# B&R Automation Studio project NAELD004C00R10L518F00 (part 14)

#### Act_OptP0934RstMnl.st
```iecst
ACTION Act_OptP0934RstMnl:

	IF EDGEPOS((bManualMod = FALSE) OR (p_eAWOpenStatus = Error)) THEN

		eAWOpenAct	:= AWActIdle;

		bJogSlow				:= FALSE;
		bJogFast				:= FALSE;
		fbJogSlowToFastDlyTm.IN	:= FALSE;

		tyP0934AW.tyAW.tyBtnGo.bRtCompl					:= FALSE;
		tyP0934AW.tyAW.tyBtnGo.bValue					:= FALSE;
		tyP0934AW.tyAW.tyBtnGo.bRtLk					:= FALSE;
		tyP0934AW.tyAW.tyBtnGo.uiMaskRtStat.0			:= FALSE;

		tyP0934AW.tyMotionStd.tyBtnPwr.bRtCompl				:= FALSE;
		tyP0934AW.tyMotionStd.tyBtnStop.bRtCompl			:= FALSE;
		tyP0934AW.tyMotionStd.tyBtnOrigin.bRtCompl			:= FALSE;
		tyP0934AW.tyMotionStd.tyBtnRst.bRtCompl				:= FALSE;
		tyP0934AW.tyMotionStd.tyBtnMovAbs.bRtCompl			:= FALSE;
		tyP0934AW.tyMotionStd.tyBtnMovRel.bRtCompl			:= FALSE;
		tyP0934AW.tyMotionStd.tyBtnJogOpen.bRtCompl			:= FALSE;
		tyP0934AW.tyMotionStd.tyBtnJogClose.bRtCompl		:= FALSE;

		tyP0934AW.tyMotionStd.tyBtnPwr.bValue				:= FALSE;
		tyP0934AW.tyMotionStd.tyBtnStop.bValue				:= TRUE;
		tyP0934AW.tyMotionStd.tyBtnOrigin.bValue			:= FALSE;
		tyP0934AW.tyMotionStd.tyBtnRst.bValue				:= FALSE;
		tyP0934AW.tyMotionStd.tyBtnMovAbs.bValue			:= FALSE;
		tyP0934AW.tyMotionStd.tyBtnMovRel.bValue			:= FALSE;
		tyP0934AW.tyMotionStd.tyBtnJogOpen.bValue			:= FALSE;
		tyP0934AW.tyMotionStd.tyBtnJogClose.bValue			:= FALSE;

		tyP0934AW.tyMotionStd.tyBtnPwr.bRtLk				:= FALSE;
		tyP0934AW.tyMotionStd.tyBtnStop.bRtLk				:= TRUE;
		tyP0934AW.tyMotionStd.tyBtnOrigin.bRtLk				:= FALSE;
		tyP0934AW.tyMotionStd.tyBtnRst.bRtLk				:= FALSE;
		tyP0934AW.tyMotionStd.tyBtnMovAbs.bRtLk				:= FALSE;
		tyP0934AW.tyMotionStd.tyBtnMovRel.bRtLk				:= FALSE;
		tyP0934AW.tyMotionStd.tyBtnJogOpen.bRtLk			:= FALSE;
		tyP0934AW.tyMotionStd.tyBtnJogClose.bRtLk			:= FALSE;

		tyP0934AW.tyMotionStd.tyBtnPwr.uiMaskRtStat			:= TRUE;
		tyP0934AW.tyMotionStd.tyBtnOrigin.uiMaskRtStat		:= FALSE;
		tyP0934AW.tyMotionStd.tyBtnRst.uiMaskRtStat			:= TRUE;
		tyP0934AW.tyMotionStd.tyBtnMovAbs.uiMaskRtStat		:= FALSE;
		tyP0934AW.tyMotionStd.tyBtnMovRel.uiMaskRtStat		:= FALSE;
		tyP0934AW.tyMotionStd.tyBtnJogOpen.uiMaskRtStat		:= FALSE;
		tyP0934AW.tyMotionStd.tyBtnJogClose.uiMaskRtStat	:= FALSE;

	END_IF

	eInShutterAct	:= PneuActIdle;
	eOutShutterAct	:= PneuActIdle;

	tyP0934AW.tyInOutletShutterFB.tyBtnClose.bRtCompl	:= FALSE;
	tyP0934AW.tyInOutletShutterFB.tyBtnClose.bValue	:= FALSE;
	tyP0934AW.tyInOutletShutterFB.tyBtnOpen.bRtCompl	:= FALSE;
	tyP0934AW.tyInOutletShutterFB.tyBtnOpen.bValue	:= FALSE;

END_ACTION
```

#### Act_OptP0934UpdtDat.st
```iecst
ACTION Act_OptP0934UpdtDat:

	tyP0934AW.tyMotionStd.tyNumCurrPos.diValue			:= p_diAWOpenActualPos;
	tyP0934AW.tyMotionStd.tyNumErrCode.diValue			:= UDINT_TO_DINT(p_udiAWOpenAxisErrID);
	tyP0934AW.tyMotionStd.tyBitmapPwr.usiValueIdx		:= BOOL_TO_USINT(p_bAWOpenPwrOn);
	tyP0934AW.tyMotionStd.tyBitmapRst.usiValueIdx		:= BOOL_TO_USINT(NOT p_bAWOpenAxisErr);
	tyP0934AW.tyMotionStd.tyBitmapOrigin.usiValueIdx	:= BOOL_TO_USINT(p_bAWOpenIsHomed);
	tyP0934AW.tyMotionStd.tyBtnOpenLmtSen.bValue		:= p_bAWOpenOpenSen;
	tyP0934AW.tyMotionStd.tyBtnCloseLmtSen.bValue		:= p_bAWOpenCloseSen;

	//Machine Bitmap //0open ,1close
	IF p_bAWOpenIsHomed = TRUE THEN
		IF p_diAWOpenActualPos <= (p_tyNtParamCurr.tyProdRcpWidth.diMax / 2) THEN
			tyP0934AW.tyMotionStd.tyBitmapMc.uiValueIdx 	:= 0;
		ELSE
			tyP0934AW.tyMotionStd.tyBitmapMc.uiValueIdx 	:= 1;
		END_IF
	ELSE
		tyP0934AW.tyMotionStd.tyBitmapMc.uiValueIdx	:= 0;
	END_IF

	IF p_tyNtParamCurr.eProjMag = LDMagTriple AND p_tyNtParamCurr.bMagAutoVerifyPrep = FALSE AND p_tyNtParamCurr.bProjMotorizedPullerPrep = FALSE AND p_tyNtParamCurr.bProjTopToBtmDefault = TRUE THEN
		IF 	tyP0934AW.tyMotionStd.tyBitmapMc.uiValueIdx < 200 THEN
			tyP0934AW.tyMotionStd.tyBitmapMc.uiValueIdx	:= tyP0934AW.tyMotionStd.tyBitmapMc.uiValueIdx + 200;
		END_IF
	ELSIF p_tyNtParamCurr.eProjMag = LDMagTriple AND p_tyNtParamCurr.bMagAutoVerifyPrep = FALSE AND p_tyNtParamCurr.bProjMotorizedPullerPrep = FALSE AND p_tyNtParamCurr.bProjTopToBtmDefault = FALSE THEN
			IF 	tyP0934AW.tyMotionStd.tyBitmapMc.uiValueIdx < 200 THEN
				tyP0934AW.tyMotionStd.tyBitmapMc.uiValueIdx	:= tyP0934AW.tyMotionStd.tyBitmapMc.uiValueIdx + 426;
			END_IF

	ELSIF p_tyNtParamCurr.eProjMag = LDMagDual AND p_tyNtParamCurr.bMagAutoVerifyPrep = FALSE THEN
		IF 	tyP0934AW.tyMotionStd.tyBitmapMc.uiValueIdx < 100 THEN
			IF p_tyNtParamCurr.sJobNo = '2023-0258A01' THEN
				tyP0934AW.tyMotionStd.tyBitmapMc.uiValueIdx	:= tyP0934AW.tyMotionStd.tyBitmapMc.uiValueIdx + 450;
			ELSIF p_tyNtParamCurr.sJobNo = '2023-0276A01' THEN
				tyP0934AW.tyMotionStd.tyBitmapMc.uiValueIdx	:= tyP0934AW.tyMotionStd.tyBitmapMc.uiValueIdx + 480;
			ELSE
				tyP0934AW.tyMotionStd.tyBitmapMc.uiValueIdx	:= tyP0934AW.tyMotionStd.tyBitmapMc.uiValueIdx + 200;
			END_IF
		END_IF
	ELSIF  p_tyNtParamCurr.bMagAutoVerifyPrep = TRUE THEN
		IF 	tyP0934AW.tyMotionStd.tyBitmapMc.uiValueIdx < 200 THEN
			tyP0934AW.tyMotionStd.tyBitmapMc.uiValueIdx	:= tyP0934AW.tyMotionStd.tyBitmapMc.uiValueIdx + 426;
		END_IF

	ELSIF p_tyNtParamCurr.eProjMag = LDMagTriple AND p_tyNtParamCurr.bMagAutoVerifyPrep = FALSE AND p_tyNtParamCurr.bProjMotorizedPullerPrep = TRUE
		AND p_tyNtParamCurr.bProjPullerRotCylPrep = FALSE THEN //fix (siemens)
		IF 	tyP0934AW.tyMotionStd.tyBitmapMc.uiValueIdx < 340 THEN
			tyP0934AW.tyMotionStd.tyBitmapMc.uiValueIdx:= tyP0934AW.tyMotionStd.tyBitmapMc.uiValueIdx + 340;
		END_IF
	ELSIF  p_tyNtParamCurr.eProjMag = LDMagTriple AND p_tyNtParamCurr.bMagAutoVerifyPrep = FALSE AND p_tyNtParamCurr.bProjMotorizedPullerPrep = TRUE
		AND p_tyNtParamCurr.bProjCurtainSenPrep = FALSE THEN
		IF 	tyP0934AW.tyMotionStd.tyBitmapMc.uiValueIdx < 300 THEN
			tyP0934AW.tyMotionStd.tyBitmapMc.uiValueIdx:= tyP0934AW.tyMotionStd.tyBitmapMc.uiValueIdx + 300;
		END_IF
	ELSIF  p_tyNtParamCurr.eProjMag = LDMagTriple AND p_tyNtParamCurr.bMagAutoVerifyPrep = FALSE AND p_tyNtParamCurr.bProjMotorizedPullerPrep = TRUE
		AND p_tyNtParamCurr.bProjCurtainSenPrep = TRUE AND p_tyNtParamCurr.bProjTopToBtmDefault = TRUE THEN
		IF 	tyP0934AW.tyMotionStd.tyBitmapMc.uiValueIdx < 365 THEN
			tyP0934AW.tyMotionStd.tyBitmapMc.uiValueIdx:= tyP0934AW.tyMotionStd.tyBitmapMc.uiValueIdx + 365;
		END_IF
	ELSIF p_tyNtParamCurr.eProjMag = LDMagTriple AND p_tyNtParamCurr.bMagAutoVerifyPrep = FALSE AND p_tyNtParamCurr.bProjMotorizedPullerPrep = TRUE
		AND p_tyNtParamCurr.bProjCurtainSenPrep = TRUE AND p_tyNtParamCurr.bProjTopToBtmDefault = FALSE THEN
		IF  tyP0934AW.tyMotionStd.tyBitmapMc.uiValueIdx < 426 THEN
			tyP0934AW.tyMotionStd.tyBitmapMc.uiValueIdx	:= tyP0934AW.tyMotionStd.tyBitmapMc.uiValueIdx + 426;
		END_IF
	END_IF
END_ACTION
```

#### Act_EntP0935Disp.st
```iecst
ACTION Act_EntP0935Disp:

	//Access Address
	p_tyC0001MotionStd ACCESS ADR(tyP0935Lifter.tyMotionStd);

	p_tyC0002FullMask ACCESS ADR(tyP0935Lifter.tyFullMaskHide);

	p_tyC0004Navi ACCESS ADR(tyP0935Lifter.tyNaviBack);

	p_tyC0005Main ACCESS ADR(tyCommon.tyMain);

	p_tyC0007Notif ACCESS ADR(tyCommon.tyNotif);

	p_tyC0008MsgBox ACCESS ADR(tyP0935Lifter.tyMsgBoxHide);

	p_tyC0009Info ACCESS ADR(tyCommon.tyInfo);

	p_tyP0935Lifter ACCESS ADR(tyP0935Lifter.tyLifter);

	//Display
	tyP0935Lifter.tyMotionStd.tyBtnPwr.bValue	:= p_bLifterBtmPwrOn;

	IF p_tyNtParamCurr.bProjLifterMagPlatform = FALSE THEN
	//	tyP0935Lifter.tyLifter.tyNumNewSlt.diValueMax	:= p_tyMagRcpCurrRcp.diTtlSlt + 1;
		tyP0935Lifter.tyLifter.tyNumNewSlt.diValueMax	:= p_tyMagRcpCurrRcp.diTtlSlt;
		tyP0935Lifter.tyLifter.tyNumNewSlt.diValueMin	:= p_tyNtParamCurr.diProjMagMinSlt;
	ELSE
		tyP0935Lifter.tyLifter.tyNumNewSlt.diValueMax	:= p_tyMagRcpCurrRcp.diTtlSlt;
		tyP0935Lifter.tyLifter.tyNumNewSlt.diValueMin	:= p_tyNtParamCurr.diProjMagMinSlt;
	END_IF

END_ACTION
```

#### Act_OptP0935FBCtrl.st
```iecst
ACTION Act_OptP0935FBCtrl:

	fbJogSlowToFastDlyTm.PT	:= T#2s;
	fbJogSlowToFastDlyTm;
	fbLmtRstTm;

	//Lifter Safety Sensor Interruption
	IF EDGENEG(p_tyDI.bLifterSafetyLmtSW1 AND p_tyDI.bLifterSafetyLmtSW2 AND p_tyDI.bLifterTimingBeltSen) THEN
		tyP0935Lifter.tyMotionStd.tyBtnStop.bRtCompl	:= TRUE;
	END_IF

//	IF EDGEPOS((p_udiLifterBtmAxisErrID = 21570 OR p_udiLifterBtmAxisErrID = 21571)
	IF EDGEPOS((p_bLifterBtmFwdLmtSen OR p_bLifterBtmRevLmtSen OR p_udiLifterBtmAxisErrID = 21570 OR p_udiLifterBtmAxisErrID = 21571)
		AND tyP0935Lifter.tyMotionStd.tyBtnJogDown.bValue = FALSE
		AND tyP0935Lifter.tyMotionStd.tyBtnJogUp.bValue = FALSE)
	THEN
		fbLmtRstTm.IN				:= TRUE;
	END_IF

	IF fbLmtRstTm.Q = TRUE THEN
		tyP0935Lifter.tyMotionStd.tyBtnRst.bRtCompl		:= TRUE;
	END_IF

	IF (tyP0935Lifter.tyMotionStd.tyBtnJogUp.bValue = FALSE AND tyP0935Lifter.tyMotionStd.tyBtnJogDown.bValue = FALSE) AND (p_bLifterBtmJogging = TRUE) THEN
		bJogStopLifter	:= TRUE;
	END_IF

	IF tyP0935Lifter.tyMotionStd.tyBtnStop.bRtCompl = TRUE THEN
		eLifterBtmAct		:= LifterActStop;

		IF p_eLifterBtmStat = LifterActStop AND p_eLifterBtmStatus = Done THEN
			eLifterBtmAct	:= LifterActIdle;

			tyP0935Lifter.tyMotionStd.tyBtnStop.bRtCompl			:= FALSE;
			tyP0935Lifter.tyMotionStd.tyBtnJogDown.bRtCompl			:= FALSE;
			tyP0935Lifter.tyMotionStd.tyBtnJogUp.bRtCompl			:= FALSE;
			tyP0935Lifter.tyMotionStd.tyBtnOrigin.bRtCompl			:= FALSE;
			tyP0935Lifter.tyMotionStd.tyBtnMovAbs.bRtCompl			:= FALSE;
			tyP0935Lifter.tyMotionStd.tyBtnMovRel.bRtCompl			:= FALSE;
			tyP0935Lifter.tyLifter.tyBtnGo.bRtCompl					:= FALSE;
			tyP0935Lifter.tyLifter.tyBtnNxtSlt.bRtCompl				:= FALSE;
			tyP0935Lifter.tyLifter.tyBtnPrevSlt.bRtCompl			:= FALSE;
			tyP0935Lifter.tyLifter.tyBtnGoLaneA.bRtCompl			:= FALSE;
			tyP0935Lifter.tyLifter.tyBtnGoLaneB.bRtCompl			:= FALSE;

			tyP0935Lifter.tyMotionStd.tyBtnStop.bValue				:= TRUE;
			tyP0935Lifter.tyMotionStd.tyBtnJogDown.bValue			:= FALSE;
			tyP0935Lifter.tyMotionStd.tyBtnJogUp.bValue				:= FALSE;
			tyP0935Lifter.tyMotionStd.tyBtnOrigin.bValue			:= FALSE;
			tyP0935Lifter.tyMotionStd.tyBtnMovAbs.bValue			:= FALSE;
			tyP0935Lifter.tyMotionStd.tyBtnMovRel.bValue			:= FALSE;
			tyP0935Lifter.tyLifter.tyBtnGo.bValue					:= FALSE;
			tyP0935Lifter.tyLifter.tyBtnNxtSlt.bValue				:= FALSE;
			tyP0935Lifter.tyLifter.tyBtnPrevSlt.bValue				:= FALSE;
			tyP0935Lifter.tyLifter.tyBtnGoLaneA.bValue				:= FALSE;
			tyP0935Lifter.tyLifter.tyBtnGoLaneB.bValue				:= FALSE;

			tyP0935Lifter.tyMotionStd.tyBtnStop.bRtLk				:= TRUE;
			tyP0935Lifter.tyMotionStd.tyBtnJogDown.bRtLk			:= FALSE;
			tyP0935Lifter.tyMotionStd.tyBtnJogUp.bRtLk				:= FALSE;
			tyP0935Lifter.tyMotionStd.tyBtnOrigin.bRtLk				:= FALSE;
			tyP0935Lifter.tyMotionStd.tyBtnMovAbs.bRtLk				:= FALSE;
			tyP0935Lifter.tyMotionStd.tyBtnMovRel.bRtLk				:= FALSE;
			tyP0935Lifter.tyLifter.tyBtnGo.bRtLk					:= FALSE;
			tyP0935Lifter.tyLifter.tyBtnNxtSlt.bRtLk				:= FALSE;
			tyP0935Lifter.tyLifter.tyBtnPrevSlt.bRtLk				:= FALSE;
			tyP0935Lifter.tyLifter.tyBtnGoLaneA.bRtLk				:= FALSE;
			tyP0935Lifter.tyLifter.tyBtnGoLaneB.bRtLk				:= FALSE;
		END_IF

	ELSIF (tyP0935Lifter.tyMotionStd.tyBtnJogDown.bRtCompl = TRUE) OR (tyP0935Lifter.tyMotionStd.tyBtnJogUp.bRtCompl = TRUE) OR (bJogStopLifter = TRUE) THEN
		bJogSlow					:= FALSE;
		bJogFast					:= FALSE;
		fbJogSlowToFastDlyTm.IN		:= FALSE;

		eLifterBtmAct		:= LifterActJogStop;

		IF p_eLifterBtmStat = LifterActJogStop AND p_eLifterBtmStatus = Done THEN
			eLifterBtmAct		:= LifterActIdle;

			bJogStopLifter	:= FALSE;

			tyP0935Lifter.tyMotionStd.tyBtnStop.bRtCompl			:= FALSE;
			tyP0935Lifter.tyMotionStd.tyBtnJogDown.bRtCompl			:= FALSE;
			tyP0935Lifter.tyMotionStd.tyBtnJogUp.bRtCompl			:= FALSE;
			tyP0935Lifter.tyMotionStd.tyBtnOrigin.bRtCompl			:= FALSE;
			tyP0935Lifter.tyMotionStd.tyBtnMovAbs.bRtCompl			:= FALSE;
			tyP0935Lifter.tyMotionStd.tyBtnMovRel.bRtCompl			:= FALSE;
			tyP0935Lifter.tyLifter.tyBtnGo.bRtCompl					:= FALSE;
			tyP0935Lifter.tyLifter.tyBtnNxtSlt.bRtCompl				:= FALSE;
			tyP0935Lifter.tyLifter.tyBtnPrevSlt.bRtCompl			:= FALSE;
			tyP0935Lifter.tyLifter.tyBtnGoLaneA.bRtCompl 			:= FALSE;
			tyP0935Lifter.tyLifter.tyBtnGoLaneB.bRtCompl 			:= FALSE;

			tyP0935Lifter.tyMotionStd.tyBtnStop.bValue				:= TRUE;
			tyP0935Lifter.tyMotionStd.tyBtnJogDown.bValue			:= FALSE;
			tyP0935Lifter.tyMotionStd.tyBtnJogUp.bValue				:= FALSE;
			tyP0935Lifter.tyMotionStd.tyBtnOrigin.bValue			:= FALSE;
			tyP0935Lifter.tyMotionStd.tyBtnMovAbs.bValue			:= FALSE;
			tyP0935Lifter.tyMotionStd.tyBtnMovRel.bValue			:= FALSE;
			tyP0935Lifter.tyLifter.tyBtnGo.bValue					:= FALSE;
			tyP0935Lifter.tyLifter.tyBtnNxtSlt.bValue				:= FALSE;
			tyP0935Lifter.tyLifter.tyBtnPrevSlt.bValue				:= FALSE;
			tyP0935Lifter.tyLifter.tyBtnGoLaneA.bValue 				:= FALSE;
			tyP0935Lifter.tyLifter.tyBtnGoLaneB.bValue 				:= FALSE;

			tyP0935Lifter.tyMotionStd.tyBtnStop.bRtLk				:= TRUE;
			tyP0935Lifter.tyMotionStd.tyBtnJogDown.bRtLk			:= FALSE;
			tyP0935Lifter.tyMotionStd.tyBtnJogUp.bRtLk				:= FALSE;
			tyP0935Lifter.tyMotionStd.tyBtnOrigin.bRtLk				:= FALSE;
			tyP0935Lifter.tyMotionStd.tyBtnMovAbs.bRtLk				:= FALSE;
			tyP0935Lifter.tyMotionStd.tyBtnMovRel.bRtLk				:= FALSE;
			tyP0935Lifter.tyLifter.tyBtnGo.bRtLk					:= FALSE;
			tyP0935Lifter.tyLifter.tyBtnNxtSlt.bRtLk				:= FALSE;
			tyP0935Lifter.tyLifter.tyBtnPrevSlt.bRtLk				:= FALSE;
			tyP0935Lifter.tyLifter.tyBtnGoLaneA.bRtLk 				:= FALSE;
			tyP0935Lifter.tyLifter.tyBtnGoLaneB.bRtLk 				:= FALSE;

		END_IF

	ELSIF tyP0935Lifter.tyMotionStd.tyBtnPwr.bRtCompl = TRUE THEN
		tyP0935Lifter.tyMotionStd.tyBtnPwr.bRtLk					:= TRUE;

		IF tyP0935Lifter.tyMotionStd.tyBtnPwr.bValue = TRUE THEN
			eLifterBtmAct		:= LifterActPwrOn;

			IF p_eLifterBtmStat = LifterActPwrOn AND p_eLifterBtmStatus = Done THEN
				eLifterBtmAct	:= LifterActIdle;

				tyP0935Lifter.tyMotionStd.tyBtnPwr.bRtCompl		:= FALSE;
				tyP0935Lifter.tyMotionStd.tyBtnPwr.bRtLk		:= FALSE;
			END_IF
		ELSE
			eLifterBtmAct		:= LifterActPwrOff;

			IF p_eLifterBtmStat = LifterActPwrOff AND p_eLifterBtmStatus = Done THEN
				eLifterBtmAct	:= LifterActIdle;

				tyP0935Lifter.tyMotionStd.tyBtnPwr.bRtCompl		:= FALSE;
				tyP0935Lifter.tyMotionStd.tyBtnPwr.bRtLk		:= FALSE;
			END_IF
		END_IF

	ELSIF tyP0935Lifter.tyMotionStd.tyBtnOrigin.bRtCompl = TRUE THEN
		tyP0935Lifter.tyMotionStd.tyBtnOrigin.bValue				:= TRUE;
		tyP0935Lifter.tyMotionStd.tyBtnStop.bValue					:= FALSE;

		tyP0935Lifter.tyMotionStd.tyBtnOrigin.bRtLk					:= TRUE;
		tyP0935Lifter.tyMotionStd.tyBtnStop.bRtLk					:= FALSE;

		eLifterBtmAct		:= LifterActHoming;

		IF p_eLifterBtmStat = LifterActHoming AND p_eLifterBtmStatus = Done THEN
			eLifterBtmAct	:= LifterActIdle;

			tyP0935Lifter.tyMotionStd.tyBtnOrigin.bRtCompl		:= FALSE;
			tyP0935Lifter.tyMotionStd.tyBtnOrigin.bValue		:= FALSE;
			tyP0935Lifter.tyMotionStd.tyBtnStop.bValue			:= TRUE;

			tyP0935Lifter.tyMotionStd.tyBtnOrigin.bRtLk			:= FALSE;
			tyP0935Lifter.tyMotionStd.tyBtnStop.bRtLk			:= TRUE;

		END_IF

	ELSIF tyP0935Lifter.tyMotionStd.tyBtnRst.bRtCompl = TRUE THEN
		tyP0935Lifter.tyMotionStd.tyBtnRst.bValue				:= TRUE;
		tyP0935Lifter.tyMotionStd.tyBtnRst.bRtLk				:= TRUE;

		eLifterBtmAct		:= LifterActRstAxisErr;

		IF p_eLifterBtmStat = LifterActRstAxisErr AND p_eLifterBtmStatus = Done THEN
			eLifterBtmAct	:= LifterActIdle;

			tyP0935Lifter.tyMotionStd.tyBtnRst.bRtCompl			:= FALSE;
			tyP0935Lifter.tyMotionStd.tyBtnRst.bValue			:= FALSE;
			tyP0935Lifter.tyMotionStd.tyBtnRst.bRtLk			:= FALSE;

			fbLmtRstTm.IN			:= FALSE;
		END_IF

	ELSIF tyP0935Lifter.tyLifter.tyBtnGo.bRtCompl = TRUE THEN
		tyP0935Lifter.tyLifter.tyBtnGo.bValue				:= TRUE;
		tyP0935Lifter.tyMotionStd.tyBtnStop.bValue			:= FALSE;

		tyP0935Lifter.tyLifter.tyBtnGo.bRtLk				:= TRUE;
		tyP0935Lifter.tyMotionStd.tyBtnStop.bRtLk			:= FALSE;

		(*diMnlLifterMag1GoSlt	:= tyP0935Lifter.tyLifter.tyNumNewSlt.diValue;*)
		diMnlLifterNomSpd		:= tyP0935Lifter.tyMotionStd.tyNumNomSpd.diValue;

		CASE tyP0935Lifter.tyLifter.tyNumMagPos.diValue OF
			1:
				eLifterBtmAct	:= LifterActGoASltPos;
				diMnlLifterMag1GoSlt	:= tyP0935Lifter.tyLifter.tyNumNewSlt.diValue;

			2:
				eLifterBtmAct	:= LifterActGoBSltPos;
				diMnlLifterMag2GoSlt	:= tyP0935Lifter.tyLifter.tyNumNewSlt.diValue;

			3:
				eLifterBtmAct	:= LifterActGoCSltPos;
				diMnlLifterMag3GoSlt	:= tyP0935Lifter.tyLifter.tyNumNewSlt.diValue;

			4:
				eLifterBtmAct	:= LifterActGoDSltPos;
				diMnlLifterMag3GoSlt	:= tyP0935Lifter.tyLifter.tyNumNewSlt.diValue;
		END_CASE

		IF (p_eLifterBtmStat = LifterActGoASltPos
			OR p_eLifterBtmStat = LifterActGoBSltPos
			OR p_eLifterBtmStat = LifterActGoCSltPos
			OR p_eLifterBtmStat = LifterActGoDSltPos)
			AND p_eLifterBtmStatus = Done THEN
			eLifterBtmAct	:= LifterActIdle;

			tyP0935Lifter.tyLifter.tyBtnGo.bRtCompl				:= FALSE;
			tyP0935Lifter.tyLifter.tyBtnGo.bValue				:= FALSE;
			tyP0935Lifter.tyMotionStd.tyBtnStop.bValue			:= TRUE;

			tyP0935Lifter.tyLifter.tyBtnGo.bRtLk				:= FALSE;
			tyP0935Lifter.tyMotionStd.tyBtnStop.bRtLk			:= TRUE;
		END_IF

	ELSIF tyP0935Lifter.tyLifter.tyBtnNxtSlt.bRtCompl = TRUE THEN
		tyP0935Lifter.tyLifter.tyBtnNxtSlt.bValue				:= TRUE;
		tyP0935Lifter.tyMotionStd.tyBtnStop.bValue				:= FALSE;

		tyP0935Lifter.tyLifter.tyBtnNxtSlt.bRtLk				:= TRUE;
		tyP0935Lifter.tyMotionStd.tyBtnStop.bRtLk				:= FALSE;

		(*diMnlLifterMag1GoSlt	:= tyP0935Lifter.tyLifter.tyNumNewSlt.diValue;*)
		diMnlLifterNomSpd		:= tyP0935Lifter.tyMotionStd.tyNumNomSpd.diValue;

		CASE tyP0935Lifter.tyLifter.tyNumMagPos.diValue OF
			1:
				eLifterBtmAct	:= LifterActGoNxtASltPos;
				diMnlLifterMag1GoSlt	:= tyP0935Lifter.tyLifter.tyNumNewSlt.diValue;
			2:
				eLifterBtmAct	:= LifterActGoNxtBSltPos;
				diMnlLifterMag2GoSlt	:= tyP0935Lifter.tyLifter.tyNumNewSlt.diValue;
			3:
				eLifterBtmAct	:= LifterActGoNxtCSltPos;
				diMnlLifterMag3GoSlt	:= tyP0935Lifter.tyLifter.tyNumNewSlt.diValue;
			4:
				eLifterBtmAct	:= LifterActGoNxtDSltPos;
				diMnlLifterMag4GoSlt	:= tyP0935Lifter.tyLifter.tyNumNewSlt.diValue;

		END_CASE

		IF (p_eLifterBtmStat = LifterActGoNxtASltPos
			OR p_eLifterBtmStat = LifterActGoNxtBSltPos
			OR p_eLifterBtmStat = LifterActGoNxtCSltPos
			OR p_eLifterBtmStat = LifterActGoNxtDSltPos)
			AND p_eLifterBtmStatus = Done THEN
			eLifterBtmAct	:= LifterActIdle;

			tyP0935Lifter.tyLifter.tyBtnNxtSlt.bRtCompl				:= FALSE;
			tyP0935Lifter.tyLifter.tyBtnNxtSlt.bValue				:= FALSE;
			tyP0935Lifter.tyMotionStd.tyBtnStop.bValue				:= TRUE;

			tyP0935Lifter.tyLifter.tyBtnNxtSlt.bRtLk				:= FALSE;
			tyP0935Lifter.tyMotionStd.tyBtnStop.bRtLk				:= TRUE;
		END_IF

	ELSIF tyP0935Lifter.tyLifter.tyBtnPrevSlt.bRtCompl = TRUE THEN
		tyP0935Lifter.tyLifter.tyBtnPrevSlt.bValue				:= TRUE;
		tyP0935Lifter.tyMotionStd.tyBtnStop.bValue				:= FALSE;

		tyP0935Lifter.tyLifter.tyBtnPrevSlt.bRtLk				:= TRUE;
		tyP0935Lifter.tyMotionStd.tyBtnStop.bRtLk				:= FALSE;

		//diMnlLifterMag1GoSlt	:= tyP0935Lifter.tyLifter.tyNumNewSlt.diValue;
		diMnlLifterNomSpd		:= tyP0935Lifter.tyMotionStd.tyNumNomSpd.diValue;

		CASE tyP0935Lifter.tyLifter.tyNumMagPos.diValue OF

			1:
				eLifterBtmAct	:= LifterActGoPrevASltPos;
				diMnlLifterMag1GoSlt	:= tyP0935Lifter.tyLifter.tyNumNewSlt.diValue;

			2:
				eLifterBtmAct	:= LifterActGoPrevBSltPos;
				diMnlLifterMag2GoSlt	:= tyP0935Lifter.tyLifter.tyNumNewSlt.diValue;

			3:
				eLifterBtmAct	:= LifterActGoPrevCSltPos;
				diMnlLifterMag3GoSlt	:= tyP0935Lifter.tyLifter.tyNumNewSlt.diValue;

			4:
				eLifterBtmAct	:= LifterActGoPrevDSltPos;
				diMnlLifterMag4GoSlt	:= tyP0935Lifter.tyLifter.tyNumNewSlt.diValue;

		END_CASE

		IF (p_eLifterBtmStat = LifterActGoPrevASltPos
			OR p_eLifterBtmStat = LifterActGoPrevBSltPos
			OR p_eLifterBtmStat = LifterActGoPrevCSltPos
			OR p_eLifterBtmStat = LifterActGoPrevDSltPos)
			AND p_eLifterBtmStatus = Done THEN
			eLifterBtmAct	:= LifterActIdle;

			tyP0935Lifter.tyLifter.tyBtnPrevSlt.bRtCompl				:= FALSE;
			tyP0935Lifter.tyLifter.tyBtnPrevSlt.bValue					:= FALSE;
			tyP0935Lifter.tyMotionStd.tyBtnStop.bValue					:= TRUE;

			tyP0935Lifter.tyLifter.tyBtnPrevSlt.bRtLk					:= FALSE;
			tyP0935Lifter.tyMotionStd.tyBtnStop.bRtLk					:= TRUE;
		END_IF

	ELSIF tyP0935Lifter.tyLifter.tyBtnGoLaneA.bRtCompl = TRUE THEN
		tyP0935Lifter.tyLifter.tyBtnGoLaneA.bValue	:= TRUE;
		tyP0935Lifter.tyMotionStd.tyBtnStop.bValue	:= FALSE;

		tyP0935Lifter.tyLifter.tyBtnGoLaneA.bRtLk	:= TRUE;
		tyP0935Lifter.tyMotionStd.tyBtnStop.bRtLk	:= FALSE;

		diMnlLifterNomSpd	:= tyP0935Lifter.tyMotionStd.tyNumNomSpd.diValue;

		eLifterBtmAct	:= LifterActGoAPos;

		IF p_eLifterBtmStat = LifterActGoAPos AND p_eLifterBtmStatus = Done THEN
			eLifterBtmAct	:= LifterActIdle;

			tyP0935Lifter.tyLifter.tyBtnGoLaneA.bRtCompl	:= FALSE;

			tyP0935Lifter.tyLifter.tyBtnGoLaneA.bValue	:= FALSE;
			tyP0935Lifter.tyMotionStd.tyBtnStop.bValue	:= TRUE;

			tyP0935Lifter.tyLifter.tyBtnGoLaneA.bRtLk	:= FALSE;
			tyP0935Lifter.tyMotionStd.tyBtnStop.bRtLk	:= TRUE;
		END_IF

	ELSIF tyP0935Lifter.tyLifter.tyBtnGoLaneB.bRtCompl = TRUE THEN
		tyP0935Lifter.tyLifter.tyBtnGoLaneB.bValue	:= TRUE;
		tyP0935Lifter.tyMotionStd.tyBtnStop.bValue	:= FALSE;

		tyP0935Lifter.tyLifter.tyBtnGoLaneB.bRtLk	:= TRUE;
		tyP0935Lifter.tyMotionStd.tyBtnStop.bRtLk	:= FALSE;

		diMnlLifterNomSpd	:= tyP0935Lifter.tyMotionStd.tyNumNomSpd.diValue;

		eLifterBtmAct	:= LifterActGoBPos;

		IF p_eLifterBtmStat = LifterActGoBPos AND p_eLifterBtmStatus = Done THEN
			eLifterBtmAct	:= LifterActIdle;

			tyP0935Lifter.tyLifter.tyBtnGoLaneB.bRtCompl	:= FALSE;

			tyP0935Lifter.tyLifter.tyBtnGoLaneB.bValue	:= FALSE;
			tyP0935Lifter.tyMotionStd.tyBtnStop.bValue	:= TRUE;

			tyP0935Lifter.tyLifter.tyBtnGoLaneB.bRtLk	:= FALSE;
			tyP0935Lifter.tyMotionStd.tyBtnStop.bRtLk	:= TRUE;
		END_IF

	ELSIF tyP0935Lifter.tyMotionStd.tyBtnMovAbs.bRtCompl = TRUE THEN

		tyP0935Lifter.tyMotionStd.tyBtnMovAbs.bValue				:= TRUE;
		tyP0935Lifter.tyMotionStd.tyBtnStop.bValue					:= FALSE;

		tyP0935Lifter.tyMotionStd.tyBtnMovAbs.bRtLk					:= TRUE;
		tyP0935Lifter.tyMotionStd.tyBtnStop.bRtLk					:= FALSE;

		diMnlLifterTargetPos	:= tyP0935Lifter.tyMotionStd.tyNumTargetPos.diValue;
		diMnlLifterNomSpd		:= tyP0935Lifter.tyMotionStd.tyNumNomSpd.diValue;

		eLifterBtmAct			:= LifterActMovAbs;

		IF p_eLifterBtmStat = LifterActMovAbs AND p_eLifterBtmStatus = Done THEN
			eLifterBtmAct	:= LifterActIdle;

			tyP0935Lifter.tyMotionStd.tyBtnMovAbs.bRtCompl		:= FALSE;
			tyP0935Lifter.tyMotionStd.tyBtnMovAbs.bValue		:= FALSE;
			tyP0935Lifter.tyMotionStd.tyBtnStop.bValue			:= TRUE;

			tyP0935Lifter.tyMotionStd.tyBtnMovAbs.bRtLk			:= FALSE;
			tyP0935Lifter.tyMotionStd.tyBtnStop.bRtLk			:= TRUE;
		END_IF

	ELSIF tyP0935Lifter.tyMotionStd.tyBtnMovRel.bRtCompl = TRUE THEN
		tyP0935Lifter.tyMotionStd.tyBtnMovRel.bValue			:= TRUE;
		tyP0935Lifter.tyMotionStd.tyBtnStop.bValue				:= FALSE;

		tyP0935Lifter.tyMotionStd.tyBtnMovRel.bRtLk				:= TRUE;
		tyP0935Lifter.tyMotionStd.tyBtnStop.bRtLk				:= FALSE;

		diMnlLifterStepSize		:= tyP0935Lifter.tyMotionStd.tyNumStepSize.diValue;
		diMnlLifterNomSpd		:= tyP0935Lifter.tyMotionStd.tyNumNomSpd.diValue;

		eLifterBtmAct		:= LifterActMovRel;

		IF p_eLifterBtmStat = LifterActMovRel AND p_eLifterBtmStatus = Done THEN
			eLifterBtmAct	:= LifterActIdle;

			tyP0935Lifter.tyMotionStd.tyBtnMovRel.bRtCompl		:= FALSE;
			tyP0935Lifter.tyMotionStd.tyBtnMovRel.bValue		:= FALSE;
			tyP0935Lifter.tyMotionStd.tyBtnStop.bValue			:= TRUE;

			tyP0935Lifter.tyMotionStd.tyBtnMovRel.bRtLk			:= FALSE;
			tyP0935Lifter.tyMotionStd.tyBtnStop.bRtLk			:= TRUE;

		END_IF

	ELSIF (tyP0935Lifter.tyMotionStd.tyBtnJogDown.bValue = TRUE) AND (fbJogSlowToFastDlyTm.Q = FALSE) AND (bJogSlow = FALSE) THEN
		tyP0935Lifter.tyMotionStd.tyBtnStop.bValue				:= FALSE;
		tyP0935Lifter.tyMotionStd.tyBtnStop.bRtLk				:= FALSE;

		fbJogSlowToFastDlyTm.IN		:= TRUE;

		diMnlLifterJogSpd	:= tyP0935Lifter.tyMotionStd.tyNumSlwSpd.diValue;

		eLifterBtmAct		:= LifterActJogDown;

		IF p_eLifterBtmStat = LifterActJogDown AND p_eLifterBtmStatus = Done THEN

			eLifterBtmAct	:= LifterActIdle;
			bJogSlow				:= TRUE;

		ELSIF p_eLifterBtmStatus = Error THEN

			fbJogSlowToFastDlyTm.IN	:= FALSE;
			bJogSlow				:= TRUE;

		END_IF

	ELSIF (tyP0935Lifter.tyMotionStd.tyBtnJogDown.bValue = TRUE) AND (fbJogSlowToFastDlyTm.Q = TRUE) AND (bJogFast = FALSE) THEN
		tyP0935Lifter.tyMotionStd.tyBtnStop.bValue					:= FALSE;
		tyP0935Lifter.tyMotionStd.tyBtnStop.bRtLk					:= FALSE;

		fbJogSlowToFastDlyTm.IN		:= TRUE;

		diMnlLifterJogSpd	:= tyP0935Lifter.tyMotionStd.tyNumNomSpd.diValue;

		eLifterBtmAct		:= LifterActJogDown;

		IF p_eLifterBtmStat = LifterActJogDown AND p_eLifterBtmStatus = Done THEN
			eLifterBtmAct	:= LifterActIdle;
			bJogFast				:= TRUE;
		ELSIF p_eLifterBtmStatus = Error THEN
			fbJogSlowToFastDlyTm.IN	:= FALSE;
			bJogFast				:= TRUE;
		END_IF

	ELSIF (tyP0935Lifter.tyMotionStd.tyBtnJogUp.bValue = TRUE) AND (fbJogSlowToFastDlyTm.Q = FALSE) AND (bJogSlow = FALSE) THEN
		tyP0935Lifter.tyMotionStd.tyBtnStop.bValue				:= FALSE;
		tyP0935Lifter.tyMotionStd.tyBtnStop.bRtLk				:= FALSE;

		fbJogSlowToFastDlyTm.IN		:= TRUE;

		diMnlLifterJogSpd	:= tyP0935Lifter.tyMotionStd.tyNumSlwSpd.diValue;

		eLifterBtmAct		:= LifterActJogUp;

		IF p_eLifterBtmStat = LifterActJogUp AND p_eLifterBtmStatus = Done THEN
			eLifterBtmAct	:= LifterActIdle;
			bJogSlow				:= TRUE;

		ELSIF p_eLifterBtmStatus = Error THEN
			fbJogSlowToFastDlyTm.IN	:= FALSE;
			bJogSlow				:= TRUE;
		END_IF

	ELSIF (tyP0935Lifter.tyMotionStd.tyBtnJogUp.bValue = TRUE) AND (fbJogSlowToFastDlyTm.Q = TRUE) AND (bJogFast = FALSE) THEN

		tyP0935Lifter.tyMotionStd.tyBtnStop.bValue				:= FALSE;
		tyP0935Lifter.tyMotionStd.tyBtnStop.bRtLk				:= FALSE;

		fbJogSlowToFastDlyTm.IN		:= TRUE;

		diMnlLifterJogSpd	:= tyP0935Lifter.tyMotionStd.tyNumNomSpd.diValue;

		eLifterBtmAct		:= LifterActJogUp;

		IF p_eLifterBtmStat = LifterActJogUp AND p_eLifterBtmStatus = Done THEN
			eLifterBtmAct	:= LifterActIdle;
			bJogFast	:= TRUE;

		ELSIF p_eLifterBtmStatus = Error THEN
			fbJogSlowToFastDlyTm.IN	:= FALSE;
			bJogFast				:= TRUE;
		END_IF
	END_IF

	//Shutter Control
	IF tyP0935Lifter.tyInOutletShutterFB.tyBtnOpen.bRtCompl = TRUE THEN
		tyP0935Lifter.tyInOutletShutterFB.tyBtnOpen.bRtCompl	:= FALSE;

		tyP0935Lifter.tyInOutletShutterFB.tyBtnOpen.bValue	:= TRUE;
		tyP0935Lifter.tyInOutletShutterFB.tyBtnClose.bValue	:= FALSE;

	ELSIF tyP0935Lifter.tyInOutletShutterFB.tyBtnClose.bRtCompl = TRUE THEN
		tyP0935Lifter.tyInOutletShutterFB.tyBtnClose.bRtCompl	:= FALSE;

		tyP0935Lifter.tyInOutletShutterFB.tyBtnClose.bValue	:= TRUE;
		tyP0935Lifter.tyInOutletShutterFB.tyBtnOpen.bValue	:= FALSE;
	END_IF

	IF tyP0935Lifter.tyInOutletShutterFB.tyBtnOpen.bValue = TRUE THEN
		eInShutterAct	:= PneuActRet;
		eOutShutterAct	:= PneuActRet;

		IF (p_eInShutterStat = PneuActRet AND p_eInShutterStatus = Done)
			AND (p_eOutShutterStat = PneuActRet AND p_eOutShutterStatus = Done)
			THEN
			eInShutterAct	:= PneuActIdle;
			eOutShutterAct	:= PneuActIdle;
			tyP0935Lifter.tyInOutletShutterFB.tyBtnOpen.bValue	:= FALSE;
		ELSIF p_eInShutterStatus = Error OR p_eOutShutterStatus = Error THEN
			tyP0935Lifter.tyInOutletShutterFB.tyBtnOpen.bValue	:= FALSE;
		END_IF

	ELSIF tyP0935Lifter.tyInOutletShutterFB.tyBtnClose.bValue = TRUE THEN
		eInShutterAct	:= PneuActExt;
		eOutShutterAct	:= PneuActExt;
		IF (p_eInShutterStat = PneuActExt AND p_eInShutterStatus = Done)
			AND (p_eOutShutterStat = PneuActExt AND p_eOutShutterStatus = Done)
			THEN
			eInShutterAct	:= PneuActIdle;
			eOutShutterAct	:= PneuActIdle;
			tyP0935Lifter.tyInOutletShutterFB.tyBtnClose.bValue := FALSE;
		ELSIF p_eInShutterStatus = Error OR p_eOutShutterStatus = Error THEN
			tyP0935Lifter.tyInOutletShutterFB.tyBtnClose.bValue := FALSE;
		END_IF
	END_IF

END_ACTION
```

#### Act_OptP0935FullMask.st
```iecst
ACTION Act_OptP0935FullMask:

	IF eCurrPage = UIP0935Lifter THEN

		IF p_tyDI.bEStopSig = FALSE THEN
			p_tyC0002FullMask ACCESS ADR(tyP0935Lifter.tyFullMaskEStop);

		ELSIF p_tyDI.bCoverSWSig = FALSE THEN
			p_tyC0002FullMask ACCESS ADR(tyP0935Lifter.tyFullMaskCWSig);

		ELSIF p_tyDI.bSafetyRlySig = FALSE THEN
			p_tyC0002FullMask ACCESS ADR(tyP0935Lifter.tyFullMaskSafetyRly);

		ELSIF p_tyDI.bPullerRetRS = FALSE THEN
			p_tyC0002FullMask ACCESS ADR(tyP0935Lifter.tyFullMaskPullInterrupt);

		ELSIF p_tyNtParamCurr.bProjInletShutPrep AND (p_tyDI.bInShutterCloseRS = FALSE
			OR (p_tyDI.bInShutterCloseRS2 = FALSE AND p_tyNtParamCurr.tyDISettings.diInShutterCloseRS2 > 0)
			OR (p_tyDI.bInShutterCloseRS3 = FALSE AND p_tyNtParamCurr.tyDISettings.diInShutterCloseRS3 > 0)) THEN
			IF p_tyNtParamCurr.bProjCurtainSenPrep THEN
				IF p_tyDI.bInShutterCloseRS = FALSE OR p_tyDI.bInShutterCloseRS2 = FALSE OR p_tyDI.bInShutterCloseRS3 = FALSE THEN
					p_tyC0002FullMask ACCESS ADR(tyP0935Lifter.tyFullMaskInShutOpnInterrupt);
				END_IF
			ELSE
				IF p_tyDI.bInShutterCloseRS = FALSE THEN
					p_tyC0002FullMask ACCESS ADR(tyP0935Lifter.tyFullMaskInShutOpnInterrupt);
				END_IF
			END_IF

	//	ELSIF p_tyNtParamCurr.bProjOutletShutPrep AND p_tyDI.bOutShutterCloseRS = FALSE AND p_McParamOutShutterDis = FALSE THEN
		ELSIF p_tyNtParamCurr.bProjOutletShutPrep AND p_tyDI.bOutShutterCloseRS = FALSE THEN
			p_tyC0002FullMask ACCESS ADR(tyP0935Lifter.tyFullMaskOutShutOpnInterrupt);

		ELSIF p_tyDI.bConvLftSen THEN
			p_tyC0002FullMask ACCESS ADR(tyP0935Lifter.tyFullMaskLftSenInterrupt);

		ELSIF p_tyDI.bConvRgtSen THEN
			p_tyC0002FullMask ACCESS ADR(tyP0935Lifter.tyFullMaskRgtSenInterrupt);

		ELSIF p_tyDI.bLifterSafetyLmtSW1 = FALSE OR p_tyDI.bLifterSafetyLmtSW2 = FALSE THEN
			p_tyC0002FullMask ACCESS ADR(tyP0935Lifter.tyFullMaskSafetyLmtSW);

		ELSIF p_tyDI.bLifterTimingBeltSen = FALSE THEN
			p_tyC0002FullMask ACCESS ADR(tyP0935Lifter.tyFullMaskTimingBelt);

		ELSE
			p_tyC0002FullMask ACCESS ADR(tyP0935Lifter.tyFullMaskHide);

		END_IF

	END_IF

END_ACTION
```

#### Act_OptP0935Keypad.st
```iecst
ACTION Act_OptP0935Keypad:

	IF fUIOutRtStatTPIsOpen(ADR(tyP0935Lifter.tyMotionStd.tyNumTargetPos.uiRtStat)) = TRUE THEN
		tyProperty.tyKeypad.tyStringTitle.sKeypadTitle	:= tyP0935Lifter.tyMotionStd.tyNumTargetPos.sKeypadTitle;

	ELSIF fUIOutRtStatTPIsOpen(ADR(tyP0935Lifter.tyMotionStd.tyNumStepSize.uiRtStat)) = TRUE THEN
		tyProperty.tyKeypad.tyStringTitle.sKeypadTitle	:= tyP0935Lifter.tyMotionStd.tyNumStepSize.sKeypadTitle;

	ELSIF fUIOutRtStatTPIsOpen(ADR(tyP0935Lifter.tyMotionStd.tyNumNomSpd.uiRtStat)) = TRUE THEN
		tyProperty.tyKeypad.tyStringTitle.sKeypadTitle	:= tyP0935Lifter.tyMotionStd.tyNumNomSpd.sKeypadTitle;

	ELSIF fUIOutRtStatTPIsOpen(ADR(tyP0935Lifter.tyMotionStd.tyNumSlwSpd.uiRtStat)) = TRUE THEN
		tyProperty.tyKeypad.tyStringTitle.sKeypadTitle	:= tyP0935Lifter.tyMotionStd.tyNumSlwSpd.sKeypadTitle;

	ELSIF fUIOutRtStatTPIsOpen(ADR(tyP0935Lifter.tyLifter.tyNumNewSlt.uiRtStat)) = TRUE THEN
		tyProperty.tyKeypad.tyStringTitle.sKeypadTitle	:= tyP0935Lifter.tyLifter.tyNumNewSlt.sKeypadTitle;

	ELSIF fUIOutRtStatTPIsOpen(ADR(tyP0935Lifter.tyLifter.tyNumMagPos.uiRtStat)) = TRUE THEN
		tyProperty.tyKeypad.tyStringTitle.sKeypadTitle	:= tyP0935Lifter.tyLifter.tyNumMagPos.sKeypadTitle;

	END_IF

END_ACTION
```

#### Act_OptP0935Mask.st
```iecst
ACTION Act_OptP0935Mask:

	// Interlock Power
	IF p_bLifterBtmAxisErr = TRUE AND p_bLifterBtmPwrOn = FALSE THEN
		fUIInRtStatOff(ADR(tyP0935Lifter.tyMotionStd.tyBtnPwr.uiMaskRtStat));
		tyP0935Lifter.tyMotionStd.tyBtnPwr.bValue		:= FALSE;
	ELSE
		fUIInRtStatHide(ADR(tyP0935Lifter.tyMotionStd.tyBtnPwr.uiMaskRtStat));
	END_IF

	// Interlock Others Move
	IF p_bLifterBtmAxisErr = TRUE OR p_bLifterBtmPwrOn = FALSE THEN
		fUIInRtStatOff(ADR(tyP0935Lifter.tyMotionStd.tyBtnOrigin.uiMaskRtStat));
		fUIInRtStatOff(ADR(tyP0935Lifter.tyMotionStd.tyBtnMovRel.uiMaskRtStat));
		fUIInRtStatOff(ADR(tyP0935Lifter.tyMotionStd.tyBtnJogUp.uiMaskRtStat));
		fUIInRtStatOff(ADR(tyP0935Lifter.tyMotionStd.tyBtnJogDown.uiMaskRtStat));
	ELSE
		fUIInRtStatHide(ADR(tyP0935Lifter.tyMotionStd.tyBtnOrigin.uiMaskRtStat));
		fUIInRtStatHide(ADR(tyP0935Lifter.tyMotionStd.tyBtnMovRel.uiMaskRtStat));
		fUIInRtStatHide(ADR(tyP0935Lifter.tyMotionStd.tyBtnJogUp.uiMaskRtStat));
		fUIInRtStatHide(ADR(tyP0935Lifter.tyMotionStd.tyBtnJogDown.uiMaskRtStat));
	END_IF

	// Interlock Move Absolute
	IF p_bLifterBtmAxisErr = TRUE OR p_bLifterBtmPwrOn = FALSE OR p_bLifterBtmIsHomed = FALSE THEN

		fUIInRtStatOff(ADR(tyP0935Lifter.tyMotionStd.tyBtnMovAbs.uiMaskRtStat));

		fUIInRtStatOff(ADR(tyP0935Lifter.tyLifter.tyBtnGo.uiMaskRtStat));
		fUIInRtStatOff(ADR(tyP0935Lifter.tyLifter.tyBtnNxtSlt.uiMaskRtStat));
		fUIInRtStatOff(ADR(tyP0935Lifter.tyLifter.tyBtnPrevSlt.uiMaskRtStat));
		fUIInRtStatOff(ADR(tyP0935Lifter.tyLifter.tyBtnGoLaneA.uiMaskRtStat));
		fUIInRtStatOff(ADR(tyP0935Lifter.tyLifter.tyBtnGoLaneB.uiMaskRtStat));

	ELSE
		fUIInRtStatHide(ADR(tyP0935Lifter.tyMotionStd.tyBtnMovAbs.uiMaskRtStat));

		fUIInRtStatHide(ADR(tyP0935Lifter.tyLifter.tyBtnGo.uiMaskRtStat));
		fUIInRtStatHide(ADR(tyP0935Lifter.tyLifter.tyBtnNxtSlt.uiMaskRtStat));
		fUIInRtStatHide(ADR(tyP0935Lifter.tyLifter.tyBtnPrevSlt.uiMaskRtStat));
		fUIInRtStatHide(ADR(tyP0935Lifter.tyLifter.tyBtnGoLaneA.uiMaskRtStat));
		fUIInRtStatHide(ADR(tyP0935Lifter.tyLifter.tyBtnGoLaneB.uiMaskRtStat));

	END_IF

	//Interlock Limit Sensor
	IF tyP0935Lifter.tyMotionStd.tyBtnDownLmtSen.bValue = TRUE THEN
		fUIInRtStatOff(ADR(tyP0935Lifter.tyMotionStd.tyBtnJogDown.uiMaskRtStat));
	END_IF

	IF tyP0935Lifter.tyMotionStd.tyBtnUpLmtSen.bValue = TRUE THEN
		fUIInRtStatOff(ADR(tyP0935Lifter.tyMotionStd.tyBtnJogUp.uiMaskRtStat));
	END_IF

	// Interlock When Moving
	IF tyP0935Lifter.tyMotionStd.tyBtnOrigin.bRtCompl = TRUE THEN

		fUIInRtStatOff(ADR(tyP0935Lifter.tyMotionStd.tyBtnMovAbs.uiMaskRtStat));
		fUIInRtStatOff(ADR(tyP0935Lifter.tyMotionStd.tyBtnMovRel.uiMaskRtStat));
		fUIInRtStatOff(ADR(tyP0935Lifter.tyMotionStd.tyBtnJogUp.uiMaskRtStat));
		fUIInRtStatOff(ADR(tyP0935Lifter.tyMotionStd.tyBtnJogDown.uiMaskRtStat));

		fUIInRtStatOff(ADR(tyP0935Lifter.tyLifter.tyBtnGo.uiMaskRtStat));
		fUIInRtStatOff(ADR(tyP0935Lifter.tyLifter.tyBtnPrevSlt.uiMaskRtStat));
		fUIInRtStatOff(ADR(tyP0935Lifter.tyLifter.tyBtnNxtSlt.uiMaskRtStat));
		fUIInRtStatOff(ADR(tyP0935Lifter.tyLifter.tyBtnGoLaneA.uiMaskRtStat));
		fUIInRtStatOff(ADR(tyP0935Lifter.tyLifter.tyBtnGoLaneB.uiMaskRtStat));

	ELSIF tyP0935Lifter.tyMotionStd.tyBtnMovAbs.bRtCompl = TRUE THEN

		fUIInRtStatOff(ADR(tyP0935Lifter.tyMotionStd.tyBtnOrigin.uiMaskRtStat));
		fUIInRtStatOff(ADR(tyP0935Lifter.tyMotionStd.tyBtnMovRel.uiMaskRtStat));
		fUIInRtStatOff(ADR(tyP0935Lifter.tyMotionStd.tyBtnJogUp.uiMaskRtStat));
		fUIInRtStatOff(ADR(tyP0935Lifter.tyMotionStd.tyBtnJogDown.uiMaskRtStat));

		fUIInRtStatOff(ADR(tyP0935Lifter.tyLifter.tyBtnGo.uiMaskRtStat));
		fUIInRtStatOff(ADR(tyP0935Lifter.tyLifter.tyBtnPrevSlt.uiMaskRtStat));
		fUIInRtStatOff(ADR(tyP0935Lifter.tyLifter.tyBtnNxtSlt.uiMaskRtStat));
		fUIInRtStatOff(ADR(tyP0935Lifter.tyLifter.tyBtnGoLaneA.uiMaskRtStat));
		fUIInRtStatOff(ADR(tyP0935Lifter.tyLifter.tyBtnGoLaneB.uiMaskRtStat));

	ELSIF tyP0935Lifter.tyMotionStd.tyBtnMovRel.bRtCompl = TRUE THEN

		fUIInRtStatOff(ADR(tyP0935Lifter.tyMotionStd.tyBtnOrigin.uiMaskRtStat));
		fUIInRtStatOff(ADR(tyP0935Lifter.tyMotionStd.tyBtnMovAbs.uiMaskRtStat));
		fUIInRtStatOff(ADR(tyP0935Lifter.tyMotionStd.tyBtnJogUp.uiMaskRtStat));
		fUIInRtStatOff(ADR(tyP0935Lifter.tyMotionStd.tyBtnJogDown.uiMaskRtStat));

		fUIInRtStatOff(ADR(tyP0935Lifter.tyLifter.tyBtnGo.uiMaskRtStat));
		fUIInRtStatOff(ADR(tyP0935Lifter.tyLifter.tyBtnNxtSlt.uiMaskRtStat));
		fUIInRtStatOff(ADR(tyP0935Lifter.tyLifter.tyBtnPrevSlt.uiMaskRtStat));
		fUIInRtStatOff(ADR(tyP0935Lifter.tyLifter.tyBtnGoLaneA.uiMaskRtStat));
		fUIInRtStatOff(ADR(tyP0935Lifter.tyLifter.tyBtnGoLaneB.uiMaskRtStat));

	ELSIF tyP0935Lifter.tyMotionStd.tyBtnJogDown.bRtCompl = TRUE OR tyP0935Lifter.tyMotionStd.tyBtnJogDown.bValue = TRUE THEN
		fUIInRtStatOff(ADR(tyP0935Lifter.tyMotionStd.tyBtnOrigin.uiMaskRtStat));
		fUIInRtStatOff(ADR(tyP0935Lifter.tyMotionStd.tyBtnMovAbs.uiMaskRtStat));
		fUIInRtStatOff(ADR(tyP0935Lifter.tyMotionStd.tyBtnMovRel.uiMaskRtStat));
		fUIInRtStatOff(ADR(tyP0935Lifter.tyMotionStd.tyBtnJogUp.uiMaskRtStat));

		fUIInRtStatOff(ADR(tyP0935Lifter.tyLifter.tyBtnGo.uiMaskRtStat));
		fUIInRtStatOff(ADR(tyP0935Lifter.tyLifter.tyBtnNxtSlt.uiMaskRtStat));
		fUIInRtStatOff(ADR(tyP0935Lifter.tyLifter.tyBtnPrevSlt.uiMaskRtStat));
		fUIInRtStatOff(ADR(tyP0935Lifter.tyLifter.tyBtnGoLaneA.uiMaskRtStat));
		fUIInRtStatOff(ADR(tyP0935Lifter.tyLifter.tyBtnGoLaneB.uiMaskRtStat));

	ELSIF tyP0935Lifter.tyMotionStd.tyBtnJogUp.bRtCompl = TRUE OR tyP0935Lifter.tyMotionStd.tyBtnJogUp.bValue = TRUE THEN
		fUIInRtStatOff(ADR(tyP0935Lifter.tyMotionStd.tyBtnOrigin.uiMaskRtStat));
		fUIInRtStatOff(ADR(tyP0935Lifter.tyMotionStd.tyBtnMovAbs.uiMaskRtStat));
		fUIInRtStatOff(ADR(tyP0935Lifter.tyMotionStd.tyBtnMovRel.uiMaskRtStat));
		fUIInRtStatOff(ADR(tyP0935Lifter.tyMotionStd.tyBtnJogDown.uiMaskRtStat));

		fUIInRtStatOff(ADR(tyP0935Lifter.tyLifter.tyBtnGo.uiMaskRtStat));
		fUIInRtStatOff(ADR(tyP0935Lifter.tyLifter.tyBtnNxtSlt.uiMaskRtStat));
		fUIInRtStatOff(ADR(tyP0935Lifter.tyLifter.tyBtnPrevSlt.uiMaskRtStat));
		fUIInRtStatOff(ADR(tyP0935Lifter.tyLifter.tyBtnGoLaneA.uiMaskRtStat));
		fUIInRtStatOff(ADR(tyP0935Lifter.tyLifter.tyBtnGoLaneB.uiMaskRtStat));

	ELSIF tyP0935Lifter.tyLifter.tyBtnGo.bRtCompl = TRUE THEN
		fUIInRtStatOff(ADR(tyP0935Lifter.tyMotionStd.tyBtnOrigin.uiMaskRtStat));
		fUIInRtStatOff(ADR(tyP0935Lifter.tyMotionStd.tyBtnMovAbs.uiMaskRtStat));
		fUIInRtStatOff(ADR(tyP0935Lifter.tyMotionStd.tyBtnMovRel.uiMaskRtStat));
		fUIInRtStatOff(ADR(tyP0935Lifter.tyMotionStd.tyBtnJogUp.uiMaskRtStat));
		fUIInRtStatOff(ADR(tyP0935Lifter.tyMotionStd.tyBtnJogDown.uiMaskRtStat));

		fUIInRtStatOff(ADR(tyP0935Lifter.tyLifter.tyBtnNxtSlt.uiMaskRtStat));
		fUIInRtStatOff(ADR(tyP0935Lifter.tyLifter.tyBtnPrevSlt.uiMaskRtStat));
		fUIInRtStatOff(ADR(tyP0935Lifter.tyLifter.tyBtnGoLaneA.uiMaskRtStat));
		fUIInRtStatOff(ADR(tyP0935Lifter.tyLifter.tyBtnGoLaneB.uiMaskRtStat));

	ELSIF tyP0935Lifter.tyLifter.tyBtnNxtSlt.bRtCompl = TRUE THEN
		fUIInRtStatOff(ADR(tyP0935Lifter.tyMotionStd.tyBtnOrigin.uiMaskRtStat));
		fUIInRtStatOff(ADR(tyP0935Lifter.tyMotionStd.tyBtnMovAbs.uiMaskRtStat));
		fUIInRtStatOff(ADR(tyP0935Lifter.tyMotionStd.tyBtnMovRel.uiMaskRtStat));
		fUIInRtStatOff(ADR(tyP0935Lifter.tyMotionStd.tyBtnJogUp.uiMaskRtStat));
		fUIInRtStatOff(ADR(tyP0935Lifter.tyMotionStd.tyBtnJogDown.uiMaskRtStat));

		fUIInRtStatOff(ADR(tyP0935Lifter.tyLifter.tyBtnGo.uiMaskRtStat));
		fUIInRtStatOff(ADR(tyP0935Lifter.tyLifter.tyBtnPrevSlt.uiMaskRtStat));
		fUIInRtStatOff(ADR(tyP0935Lifter.tyLifter.tyBtnGoLaneA.uiMaskRtStat));
		fUIInRtStatOff(ADR(tyP0935Lifter.tyLifter.tyBtnGoLaneB.uiMaskRtStat));

	ELSIF tyP0935Lifter.tyLifter.tyBtnPrevSlt.bRtCompl = TRUE THEN
		fUIInRtStatOff(ADR(tyP0935Lifter.tyMotionStd.tyBtnOrigin.uiMaskRtStat));
		fUIInRtStatOff(ADR(tyP0935Lifter.tyMotionStd.tyBtnMovAbs.uiMaskRtStat));
		fUIInRtStatOff(ADR(tyP0935Lifter.tyMotionStd.tyBtnMovRel.uiMaskRtStat));
		fUIInRtStatOff(ADR(tyP0935Lifter.tyMotionStd.tyBtnJogUp.uiMaskRtStat));
		fUIInRtStatOff(ADR(tyP0935Lifter.tyMotionStd.tyBtnJogDown.uiMaskRtStat));

		fUIInRtStatOff(ADR(tyP0935Lifter.tyLifter.tyBtnGo.uiMaskRtStat));
		fUIInRtStatOff(ADR(tyP0935Lifter.tyLifter.tyBtnNxtSlt.uiMaskRtStat));
		fUIInRtStatOff(ADR(tyP0935Lifter.tyLifter.tyBtnGoLaneA.uiMaskRtStat));
		fUIInRtStatOff(ADR(tyP0935Lifter.tyLifter.tyBtnGoLaneB.uiMaskRtStat));

	ELSIF tyP0935Lifter.tyLifter.tyBtnGoLaneA.bRtCompl = TRUE THEN
		fUIInRtStatOff(ADR(tyP0935Lifter.tyMotionStd.tyBtnOrigin.uiMaskRtStat));
		fUIInRtStatOff(ADR(tyP0935Lifter.tyMotionStd.tyBtnMovAbs.uiMaskRtStat));
		fUIInRtStatOff(ADR(tyP0935Lifter.tyMotionStd.tyBtnMovRel.uiMaskRtStat));
		fUIInRtStatOff(ADR(tyP0935Lifter.tyMotionStd.tyBtnJogUp.uiMaskRtStat));
		fUIInRtStatOff(ADR(tyP0935Lifter.tyMotionStd.tyBtnJogDown.uiMaskRtStat));

		fUIInRtStatOff(ADR(tyP0935Lifter.tyLifter.tyBtnGo.uiMaskRtStat));
		fUIInRtStatOff(ADR(tyP0935Lifter.tyLifter.tyBtnNxtSlt.uiMaskRtStat));
		fUIInRtStatOff(ADR(tyP0935Lifter.tyLifter.tyBtnPrevSlt.uiMaskRtStat));
		fUIInRtStatOff(ADR(tyP0935Lifter.tyLifter.tyBtnGoLaneB.uiMaskRtStat));

	ELSIF tyP0935Lifter.tyLifter.tyBtnGoLaneB.bRtCompl = TRUE THEN
		fUIInRtStatOff(ADR(tyP0935Lifter.tyMotionStd.tyBtnOrigin.uiMaskRtStat));
		fUIInRtStatOff(ADR(tyP0935Lifter.tyMotionStd.tyBtnMovAbs.uiMaskRtStat));
		fUIInRtStatOff(ADR(tyP0935Lifter.tyMotionStd.tyBtnMovRel.uiMaskRtStat));
		fUIInRtStatOff(ADR(tyP0935Lifter.tyMotionStd.tyBtnJogUp.uiMaskRtStat));
		fUIInRtStatOff(ADR(tyP0935Lifter.tyMotionStd.tyBtnJogDown.uiMaskRtStat));

		fUIInRtStatOff(ADR(tyP0935Lifter.tyLifter.tyBtnGo.uiMaskRtStat));
		fUIInRtStatOff(ADR(tyP0935Lifter.tyLifter.tyBtnNxtSlt.uiMaskRtStat));
		fUIInRtStatOff(ADR(tyP0935Lifter.tyLifter.tyBtnPrevSlt.uiMaskRtStat));
		fUIInRtStatOff(ADR(tyP0935Lifter.tyLifter.tyBtnGoLaneA.uiMaskRtStat));

	END_IF

	//Axis Error
	IF tyP0935Lifter.tyMotionStd.tyBtnPwr.bRtCompl = TRUE THEN
		fUIInRtStatOff(ADR(tyP0935Lifter.tyMotionStd.tyBtnRst.uiMaskRtStat));
	ELSE
		fUIInRtStatHide(ADR(tyP0935Lifter.tyMotionStd.tyBtnRst.uiMaskRtStat));
	END_IF

	//Next Slot
	IF p_diLifterBtmCurrSltA >= p_tyProdRcpCurrRcp0.diMaxSltValue THEN
		fUIInRtStatOff(ADR(tyP0935Lifter.tyLifter.tyBtnNxtSlt.uiMaskRtStat));
	END_IF

	//Previous Slot
	IF p_diLifterBtmCurrSltA <= p_tyProdRcpCurrRcp0.diMinSltValue THEN
		fUIInRtStatOff(ADR(tyP0935Lifter.tyLifter.tyBtnPrevSlt.uiMaskRtStat));
	END_IF

END_ACTION
```

#### Act_OptP0935RstMnl.st
```iecst
ACTION Act_OptP0935RstMnl:

	IF EDGEPOS((bManualMod = FALSE) OR (p_eLifterBtmStatus = Error)) THEN

		eLifterBtmAct	:= LifterActIdle;

		bJogSlow				:= FALSE;
		bJogFast				:= FALSE;
		fbJogSlowToFastDlyTm.IN	:= FALSE;

		tyP0935Lifter.tyLifter.tyBtnGo.bRtCompl					:= FALSE;
		tyP0935Lifter.tyLifter.tyBtnNxtSlt.bRtCompl				:= FALSE;
		tyP0935Lifter.tyLifter.tyBtnPrevSlt.bRtCompl			:= FALSE;
		tyP0935Lifter.tyLifter.tyBtnGoLaneA.bRtCompl			:= FALSE;
		tyP0935Lifter.tyLifter.tyBtnGoLaneB.bRtCompl			:= FALSE;

		tyP0935Lifter.tyLifter.tyBtnGo.bValue					:= FALSE;
		tyP0935Lifter.tyLifter.tyBtnNxtSlt.bValue				:= FALSE;
		tyP0935Lifter.tyLifter.tyBtnPrevSlt.bValue				:= FALSE;
		tyP0935Lifter.tyLifter.tyBtnGoLaneA.bValue				:= FALSE;
		tyP0935Lifter.tyLifter.tyBtnGoLaneB.bValue				:= FALSE;

		tyP0935Lifter.tyLifter.tyBtnGo.bRtLk					:= FALSE;
		tyP0935Lifter.tyLifter.tyBtnNxtSlt.bRtLk				:= FALSE;
		tyP0935Lifter.tyLifter.tyBtnPrevSlt.bRtLk				:= FALSE;
		tyP0935Lifter.tyLifter.tyBtnGoLaneA.bRtLk				:= FALSE;
		tyP0935Lifter.tyLifter.tyBtnGoLaneB.bRtLk				:= FALSE;

		tyP0935Lifter.tyLifter.tyBtnGo.uiMaskRtStat.0			:= FALSE;
		tyP0935Lifter.tyLifter.tyBtnNxtSlt.uiMaskRtStat.0		:= FALSE;
		tyP0935Lifter.tyLifter.tyBtnPrevSlt.uiMaskRtStat.0		:= FALSE;
		tyP0935Lifter.tyLifter.tyBtnGoLaneA.uiMaskRtStat.0		:= FALSE;
		tyP0935Lifter.tyLifter.tyBtnGoLaneB.uiMaskRtStat.0		:= FALSE;

		tyP0935Lifter.tyMotionStd.tyBtnPwr.bRtCompl				:= FALSE;
		tyP0935Lifter.tyMotionStd.tyBtnStop.bRtCompl			:= FALSE;
		tyP0935Lifter.tyMotionStd.tyBtnOrigin.bRtCompl			:= FALSE;
		tyP0935Lifter.tyMotionStd.tyBtnRst.bRtCompl				:= FALSE;
		tyP0935Lifter.tyMotionStd.tyBtnMovAbs.bRtCompl			:= FALSE;
		tyP0935Lifter.tyMotionStd.tyBtnMovRel.bRtCompl			:= FALSE;
		tyP0935Lifter.tyMotionStd.tyBtnJogUp.bRtCompl			:= FALSE;
		tyP0935Lifter.tyMotionStd.tyBtnJogDown.bRtCompl			:= FALSE;

		tyP0935Lifter.tyMotionStd.tyBtnPwr.bValue				:= FALSE;
		tyP0935Lifter.tyMotionStd.tyBtnStop.bValue				:= TRUE;
		tyP0935Lifter.tyMotionStd.tyBtnOrigin.bValue			:= FALSE;
		tyP0935Lifter.tyMotionStd.tyBtnRst.bValue				:= FALSE;
		tyP0935Lifter.tyMotionStd.tyBtnMovAbs.bValue			:= FALSE;
		tyP0935Lifter.tyMotionStd.tyBtnMovRel.bValue			:= FALSE;
		tyP0935Lifter.tyMotionStd.tyBtnJogUp.bValue				:= FALSE;
		tyP0935Lifter.tyMotionStd.tyBtnJogDown.bValue			:= FALSE;

		tyP0935Lifter.tyMotionStd.tyBtnPwr.bRtLk				:= FALSE;
		tyP0935Lifter.tyMotionStd.tyBtnStop.bRtLk				:= TRUE;
		tyP0935Lifter.tyMotionStd.tyBtnOrigin.bRtLk				:= FALSE;
		tyP0935Lifter.tyMotionStd.tyBtnRst.bRtLk				:= FALSE;
		tyP0935Lifter.tyMotionStd.tyBtnMovAbs.bRtLk				:= FALSE;
		tyP0935Lifter.tyMotionStd.tyBtnMovRel.bRtLk				:= FALSE;
		tyP0935Lifter.tyMotionStd.tyBtnJogUp.bRtLk				:= FALSE;
		tyP0935Lifter.tyMotionStd.tyBtnJogDown.bRtLk			:= FALSE;

		tyP0935Lifter.tyMotionStd.tyBtnPwr.uiMaskRtStat			:= TRUE;
		tyP0935Lifter.tyMotionStd.tyBtnOrigin.uiMaskRtStat		:= FALSE;
		tyP0935Lifter.tyMotionStd.tyBtnRst.uiMaskRtStat			:= TRUE;
		tyP0935Lifter.tyMotionStd.tyBtnMovAbs.uiMaskRtStat		:= FALSE;
		tyP0935Lifter.tyMotionStd.tyBtnMovRel.uiMaskRtStat		:= FALSE;
		tyP0935Lifter.tyMotionStd.tyBtnJogUp.uiMaskRtStat		:= FALSE;
		tyP0935Lifter.tyMotionStd.tyBtnJogDown.uiMaskRtStat		:= FALSE;

	END_IF

	eInShutterAct	:= PneuActIdle;
	eOutShutterAct	:= PneuActIdle;

	tyP0935Lifter.tyInOutletShutterFB.tyBtnClose.bRtCompl	:= FALSE;
	tyP0935Lifter.tyInOutletShutterFB.tyBtnClose.bValue	:= FALSE;
	tyP0935Lifter.tyInOutletShutterFB.tyBtnOpen.bRtCompl	:= FALSE;
	tyP0935Lifter.tyInOutletShutterFB.tyBtnOpen.bValue	:= FALSE;

END_ACTION
```

#### Act_OptP0935UpdtDat.st
```iecst
ACTION Act_OptP0935UpdtDat:

	tyP0935Lifter.tyMotionStd.tyNumCurrPos.diValue			:= p_diLifterBtmActualPos;
	tyP0935Lifter.tyMotionStd.tyNumErrCode.diValue			:= UDINT_TO_DINT(p_udiLifterBtmAxisErrID);
	tyP0935Lifter.tyMotionStd.tyBitmapPwr.usiValueIdx		:= BOOL_TO_USINT(p_bLifterBtmPwrOn);
	tyP0935Lifter.tyMotionStd.tyBitmapRst.usiValueIdx		:= BOOL_TO_USINT(NOT p_bLifterBtmAxisErr);
	tyP0935Lifter.tyMotionStd.tyBitmapOrigin.usiValueIdx	:= BOOL_TO_USINT(p_bLifterBtmIsHomed);
	tyP0935Lifter.tyMotionStd.tyBtnUpLmtSen.bValue			:= p_bLifterBtmUpSen;
	tyP0935Lifter.tyMotionStd.tyBtnDownLmtSen.bValue		:= p_bLifterBtmDownSen;

	//Machine Bitmap //default:2dn 3mid 4top
	IF  (p_tyNtParamCurr.eProjMag = LDMagDual)
		OR (p_tyNtParamCurr.eProjMag = LDMagTriple AND p_tyNtParamCurr.bMagAutoVerifyPrep = FALSE)
		THEN
			IF p_bLifterBtmIsHomed = TRUE THEN

					IF p_diLifterBtmActualPos <= (p_tyNtParamCurr.tyUILifterTargetPos.diMax / 3) THEN
						tyP0935Lifter.tyMotionStd.tyBitmapMc.uiValueIdx 	:= 2;
					ELSIF p_diLifterBtmActualPos <= (p_tyNtParamCurr.tyUILifterTargetPos.diMax / 3 * 2) THEN
						tyP0935Lifter.tyMotionStd.tyBitmapMc.uiValueIdx 	:= 3;
					ELSE
						tyP0935Lifter.tyMotionStd.tyBitmapMc.uiValueIdx 	:= 4;
					END_IF

			ELSE
				tyP0935Lifter.tyMotionStd.tyBitmapMc.uiValueIdx	:= 2;
			END_IF

	ELSIF p_tyNtParamCurr.eProjMag = LDMagTriple AND p_tyNtParamCurr.bMagAutoVerifyPrep = TRUE
		THEN
			IF p_bLifterBtmIsHomed = TRUE THEN

				IF p_diLifterBtmActualPos <= (p_tyNtParamCurr.tyUILifterTargetPos.diMax / 3) THEN
					tyP0935Lifter.tyMotionStd.tyBitmapMc.uiValueIdx 	:= 23;
				ELSIF p_diLifterBtmActualPos <= (p_tyNtParamCurr.tyUILifterTargetPos.diMax / 3 * 2) THEN
					tyP0935Lifter.tyMotionStd.tyBitmapMc.uiValueIdx 	:= 24;
				ELSE
					tyP0935Lifter.tyMotionStd.tyBitmapMc.uiValueIdx 	:= 25;
				END_IF

			ELSE
				tyP0935Lifter.tyMotionStd.tyBitmapMc.uiValueIdx	:= 23;
		END_IF
	ELSIF p_tyNtParamCurr.eProjMag = LDMagQuadruple AND p_tyNtParamCurr.bMagAutoVerifyPrep = TRUE
		THEN
		IF p_bLifterBtmIsHomed = TRUE THEN

			IF p_diLifterBtmActualPos <= (p_tyNtParamCurr.tyUILifterTargetPos.diMax / 3) THEN
				tyP0935Lifter.tyMotionStd.tyBitmapMc.uiValueIdx 	:= 27;
			ELSIF p_diLifterBtmActualPos <= (p_tyNtParamCurr.tyUILifterTargetPos.diMax / 3 * 2) THEN
				tyP0935Lifter.tyMotionStd.tyBitmapMc.uiValueIdx 	:= 28;
			ELSE
				tyP0935Lifter.tyMotionStd.tyBitmapMc.uiValueIdx 	:= 29;
			END_IF

		ELSE
			tyP0935Lifter.tyMotionStd.tyBitmapMc.uiValueIdx	:= 27;
		END_IF
	END_IF

	IF p_tyNtParamCurr.eProjMag = LDMagTriple AND p_tyNtParamCurr.bProjLifterMagPlatform THEN
		IF 	tyP0935Lifter.tyMotionStd.tyBitmapMc.uiValueIdx < 400 THEN
			tyP0935Lifter.tyMotionStd.tyBitmapMc.uiValueIdx	:= tyP0935Lifter.tyMotionStd.tyBitmapMc.uiValueIdx + 400;
		END_IF

	ELSIF p_tyNtParamCurr.eProjMag = LDMagTriple AND p_tyNtParamCurr.bMagAutoVerifyPrep = FALSE AND p_tyNtParamCurr.bProjMotorizedPullerPrep = FALSE
		THEN
			IF 	tyP0935Lifter.tyMotionStd.tyBitmapMc.uiValueIdx < 100 THEN
				tyP0935Lifter.tyMotionStd.tyBitmapMc.uiValueIdx	:= tyP0935Lifter.tyMotionStd.tyBitmapMc.uiValueIdx + 100;
		END_IF

	ELSIF p_tyNtParamCurr.eProjMag = LDMagDual AND p_tyNtParamCurr.bMagAutoVerifyPrep = FALSE
		THEN
		IF 	tyP0935Lifter.tyMotionStd.tyBitmapMc.uiValueIdx < 100 THEN
			IF p_tyNtParamCurr.bProjLifterMagPlatform THEN
			//2,3,4//	tyP0935Lifter.tyMotionStd.tyBitmapMc.uiValueIdx	:= tyP0935Lifter.tyMotionStd.tyBitmapMc.uiValueIdx + 255;
			ELSE
				IF p_tyNtParamCurr.sJobNo = '2023-0258A01' THEN
					tyP0935Lifter.tyMotionStd.tyBitmapMc.uiValueIdx	:= tyP0935Lifter.tyMotionStd.tyBitmapMc.uiValueIdx + 444-2;
				ELSIF p_tyNtParamCurr.sJobNo = '2023-0276A01' THEN
					tyP0935Lifter.tyMotionStd.tyBitmapMc.uiValueIdx	:= tyP0935Lifter.tyMotionStd.tyBitmapMc.uiValueIdx + 474-2;
				ELSE
					tyP0935Lifter.tyMotionStd.tyBitmapMc.uiValueIdx	:= tyP0935Lifter.tyMotionStd.tyBitmapMc.uiValueIdx + 200;
				END_IF
			END_IF
		END_IF

	ELSIF (p_tyNtParamCurr.eProjMag = LDMagDual OR p_tyNtParamCurr.eProjMag = LDMagTriple)
		AND p_tyNtParamCurr.bMagAutoVerifyPrep = TRUE
		THEN
		IF 	tyP0935Lifter.tyMotionStd.tyBitmapMc.uiValueIdx < 200 THEN
			tyP0935Lifter.tyMotionStd.tyBitmapMc.uiValueIdx	:= tyP0935Lifter.tyMotionStd.tyBitmapMc.uiValueIdx + 200;
		END_IF
	ELSIF p_tyNtParamCurr.eProjMag = LDMagTriple AND p_tyNtParamCurr.bMagAutoVerifyPrep = FALSE AND p_tyNtParamCurr.bProjMotorizedPullerPrep = TRUE
		AND p_tyNtParamCurr.bProjCurtainSenPrep = FALSE THEN
		IF 	tyP0935Lifter.tyMotionStd.tyBitmapMc.uiValueIdx < 300 THEN
			tyP0935Lifter.tyMotionStd.tyBitmapMc.uiValueIdx	:= tyP0935Lifter.tyMotionStd.tyBitmapMc.uiValueIdx + 300;
		END_IF
	ELSIF p_tyNtParamCurr.eProjMag = LDMagTriple AND p_tyNtParamCurr.bMagAutoVerifyPrep = FALSE AND p_tyNtParamCurr.bProjMotorizedPullerPrep = TRUE
		AND p_tyNtParamCurr.bProjCurtainSenPrep = TRUE AND p_tyNtParamCurr.bProjTopToBtmDefault = TRUE THEN
		IF 	tyP0935Lifter.tyMotionStd.tyBitmapMc.uiValueIdx < 367-2 THEN
			tyP0935Lifter.tyMotionStd.tyBitmapMc.uiValueIdx	:= tyP0935Lifter.tyMotionStd.tyBitmapMc.uiValueIdx + 367-2;
		END_IF
	ELSIF p_tyNtParamCurr.eProjMag = LDMagTriple AND p_tyNtParamCurr.bMagAutoVerifyPrep = FALSE AND p_tyNtParamCurr.bProjMotorizedPullerPrep = TRUE
		AND p_tyNtParamCurr.bProjCurtainSenPrep = TRUE AND p_tyNtParamCurr.bProjTopToBtmDefault = FALSE  THEN
		IF 	tyP0935Lifter.tyMotionStd.tyBitmapMc.uiValueIdx < 420-2 THEN
			tyP0935Lifter.tyMotionStd.tyBitmapMc.uiValueIdx	:= tyP0935Lifter.tyMotionStd.tyBitmapMc.uiValueIdx + 420-2;
		END_IF
	END_IF

END_ACTION
```

#### Act_EntP0936Disp.st
```iecst
ACTION Act_EntP0936Disp:

	//Access Address
	p_tyC0001MotionStd ACCESS ADR(tyP0936Trav.tyMotionStd);

	p_tyC0002FullMask ACCESS ADR(tyP0936Trav.tyFullMaskHide);

	p_tyC0004Navi ACCESS ADR(tyP0936Trav.tyNaviBack);

	p_tyC0005Main ACCESS ADR(tyCommon.tyMain);

	p_tyC0007Notif ACCESS ADR(tyCommon.tyNotif);

	p_tyC0008MsgBox ACCESS ADR(tyP0936Trav.tyMsgBoxHide);

	p_tyC0009Info ACCESS ADR(tyCommon.tyInfo);

	p_tyP0936Trav ACCESS ADR(tyP0936Trav.tyTrav);

	//Display
	tyP0936Trav.tyMotionStd.tyBtnPwr.bValue	:= p_bTravPwrOn;

END_ACTION
```

#### Act_OptP0936FBCtrl.st
```iecst
ACTION Act_OptP0936FBCtrl:

	fbJogSlowToFastDlyTm.PT			:= T#2s;
	fbJogSlowToFastDlyTm;
	fbLmtRstTm;

//	IF EDGEPOS((p_udiTravAxisErrID = 21570 OR p_udiTravAxisErrID = 21571)
	IF EDGEPOS ((p_bTravFwdLmtSen OR p_bTravRevLmtSen OR p_udiTravAxisErrID = 21570 OR p_udiTravAxisErrID = 21571)
		AND tyP0936Trav.tyMotionStd.tyBtnJogRear.bValue = FALSE
		AND tyP0936Trav.tyMotionStd.tyBtnJogFront.bValue = FALSE)
	THEN
		fbLmtRstTm.IN				:= TRUE;
	END_IF

	IF fbLmtRstTm.Q = TRUE THEN
		tyP0936Trav.tyMotionStd.tyBtnRst.bRtCompl		:= TRUE;
	END_IF

	IF (tyP0936Trav.tyMotionStd.tyBtnJogFront.bValue = FALSE AND tyP0936Trav.tyMotionStd.tyBtnJogRear.bValue = FALSE) AND (p_bTravJogging = TRUE) THEN
		bJogStopTrav	:= TRUE;
	END_IF

	IF tyP0936Trav.tyMotionStd.tyBtnStop.bRtCompl = TRUE THEN
		eTravAct		:= TravActStop;

		IF p_eTravStat = TravActStop AND p_eTravStatus = Done THEN
			eTravAct	:= TravActIdle;

			tyP0936Trav.tyMotionStd.tyBtnStop.bRtCompl			:= FALSE;
			tyP0936Trav.tyMotionStd.tyBtnJogRear.bRtCompl		:= FALSE;
			tyP0936Trav.tyMotionStd.tyBtnJogFront.bRtCompl		:= FALSE;
			tyP0936Trav.tyMotionStd.tyBtnOrigin.bRtCompl		:= FALSE;
			tyP0936Trav.tyMotionStd.tyBtnMovAbs.bRtCompl		:= FALSE;
			tyP0936Trav.tyMotionStd.tyBtnMovRel.bRtCompl		:= FALSE;
			tyP0936Trav.tyTrav.tyBtnGoToLaneA.bRtCompl			:= FALSE;
			tyP0936Trav.tyTrav.tyBtnGoToLaneB.bRtCompl			:= FALSE;
			tyP0936Trav.tyTrav.tyBtnGoToMag1.bRtCompl			:= FALSE;
			tyP0936Trav.tyTrav.tyBtnGoToMag2.bRtCompl			:= FALSE;
			tyP0936Trav.tyTrav.tyBtnGoToMag3.bRtCompl			:= FALSE;
			tyP0936Trav.tyTrav.tyBtnGoToMag4.bRtCompl			:= FALSE;

			tyP0936Trav.tyMotionStd.tyBtnStop.bValue			:= TRUE;
			tyP0936Trav.tyMotionStd.tyBtnJogRear.bValue			:= FALSE;
			tyP0936Trav.tyMotionStd.tyBtnJogFront.bValue		:= FALSE;
			tyP0936Trav.tyMotionStd.tyBtnOrigin.bValue			:= FALSE;
			tyP0936Trav.tyMotionStd.tyBtnMovAbs.bValue			:= FALSE;
			tyP0936Trav.tyMotionStd.tyBtnMovRel.bValue			:= FALSE;
			tyP0936Trav.tyTrav.tyBtnGoToLaneA.bValue			:= FALSE;
			tyP0936Trav.tyTrav.tyBtnGoToLaneB.bValue			:= FALSE;
			tyP0936Trav.tyTrav.tyBtnGoToMag1.bValue				:= FALSE;
			tyP0936Trav.tyTrav.tyBtnGoToMag2.bValue				:= FALSE;
			tyP0936Trav.tyTrav.tyBtnGoToMag3.bValue				:= FALSE;
			tyP0936Trav.tyTrav.tyBtnGoToMag4.bValue				:= FALSE;

			tyP0936Trav.tyMotionStd.tyBtnStop.bRtLk				:= TRUE;
			tyP0936Trav.tyMotionStd.tyBtnJogRear.bRtLk			:= FALSE;
			tyP0936Trav.tyMotionStd.tyBtnJogFront.bRtLk			:= FALSE;
			tyP0936Trav.tyMotionStd.tyBtnOrigin.bRtLk			:= FALSE;
			tyP0936Trav.tyMotionStd.tyBtnMovAbs.bRtLk			:= FALSE;
			tyP0936Trav.tyMotionStd.tyBtnMovRel.bRtLk			:= FALSE;
			tyP0936Trav.tyTrav.tyBtnGoToLaneA.bRtLk				:= FALSE;
			tyP0936Trav.tyTrav.tyBtnGoToLaneB.bRtLk				:= FALSE;
			tyP0936Trav.tyTrav.tyBtnGoToMag1.bRtLk				:= FALSE;
			tyP0936Trav.tyTrav.tyBtnGoToMag2.bRtLk				:= FALSE;
			tyP0936Trav.tyTrav.tyBtnGoToMag3.bRtLk				:= FALSE;
			tyP0936Trav.tyTrav.tyBtnGoToMag4.bRtLk				:= FALSE;
		END_IF

	ELSIF (tyP0936Trav.tyMotionStd.tyBtnJogRear.bRtCompl = TRUE) OR (tyP0936Trav.tyMotionStd.tyBtnJogFront.bRtCompl = TRUE) OR (bJogStopTrav = TRUE) THEN
		bJogSlow					:= FALSE;
		bJogFast					:= FALSE;

		fbJogSlowToFastDlyTm.IN		:= FALSE;

		eTravAct		:= TravActJogStop;

		IF p_eTravStat = TravActJogStop AND p_eTravStatus = Done THEN
			eTravAct		:= TravActIdle;

			bJogStopTrav	:= FALSE;

			tyP0936Trav.tyMotionStd.tyBtnStop.bRtCompl			:= FALSE;
			tyP0936Trav.tyMotionStd.tyBtnJogRear.bRtCompl		:= FALSE;
			tyP0936Trav.tyMotionStd.tyBtnJogFront.bRtCompl		:= FALSE;
			tyP0936Trav.tyMotionStd.tyBtnOrigin.bRtCompl		:= FALSE;
			tyP0936Trav.tyMotionStd.tyBtnMovAbs.bRtCompl		:= FALSE;
			tyP0936Trav.tyMotionStd.tyBtnMovRel.bRtCompl		:= FALSE;
			tyP0936Trav.tyTrav.tyBtnGoToLaneA.bRtCompl			:= FALSE;
			tyP0936Trav.tyTrav.tyBtnGoToLaneB.bRtCompl			:= FALSE;
			tyP0936Trav.tyTrav.tyBtnGoToMag1.bRtCompl			:= FALSE;
			tyP0936Trav.tyTrav.tyBtnGoToMag2.bRtCompl			:= FALSE;
			tyP0936Trav.tyTrav.tyBtnGoToMag3.bRtCompl			:= FALSE;
			tyP0936Trav.tyTrav.tyBtnGoToMag4.bRtCompl			:= FALSE;

			tyP0936Trav.tyMotionStd.tyBtnStop.bValue			:= TRUE;
			tyP0936Trav.tyMotionStd.tyBtnJogRear.bValue			:= FALSE;
			tyP0936Trav.tyMotionStd.tyBtnJogFront.bValue		:= FALSE;
			tyP0936Trav.tyMotionStd.tyBtnOrigin.bValue			:= FALSE;
			tyP0936Trav.tyMotionStd.tyBtnMovAbs.bValue			:= FALSE;
			tyP0936Trav.tyMotionStd.tyBtnMovRel.bValue			:= FALSE;
			tyP0936Trav.tyTrav.tyBtnGoToLaneA.bValue			:= FALSE;
			tyP0936Trav.tyTrav.tyBtnGoToLaneB.bValue			:= FALSE;
			tyP0936Trav.tyTrav.tyBtnGoToMag1.bValue				:= FALSE;
			tyP0936Trav.tyTrav.tyBtnGoToMag2.bValue				:= FALSE;
			tyP0936Trav.tyTrav.tyBtnGoToMag3.bValue				:= FALSE;
			tyP0936Trav.tyTrav.tyBtnGoToMag4.bValue				:= FALSE;

			tyP0936Trav.tyMotionStd.tyBtnStop.bRtLk				:= TRUE;
			tyP0936Trav.tyMotionStd.tyBtnJogRear.bRtLk			:= FALSE;
			tyP0936Trav.tyMotionStd.tyBtnJogFront.bRtLk			:= FALSE;
			tyP0936Trav.tyMotionStd.tyBtnOrigin.bRtLk			:= FALSE;
			tyP0936Trav.tyMotionStd.tyBtnMovAbs.bRtLk			:= FALSE;
			tyP0936Trav.tyMotionStd.tyBtnMovRel.bRtLk			:= FALSE;
			tyP0936Trav.tyTrav.tyBtnGoToLaneA.bRtLk				:= FALSE;
			tyP0936Trav.tyTrav.tyBtnGoToLaneB.bRtLk				:= FALSE;
			tyP0936Trav.tyTrav.tyBtnGoToMag1.bRtLk				:= FALSE;
			tyP0936Trav.tyTrav.tyBtnGoToMag2.bRtLk				:= FALSE;
			tyP0936Trav.tyTrav.tyBtnGoToMag3.bRtLk				:= FALSE;
			tyP0936Trav.tyTrav.tyBtnGoToMag4.bRtLk				:= FALSE;
		END_IF

	ELSIF tyP0936Trav.tyMotionStd.tyBtnPwr.bRtCompl = TRUE THEN
		tyP0936Trav.tyMotionStd.tyBtnPwr.bRtLk					:= TRUE;

		IF tyP0936Trav.tyMotionStd.tyBtnPwr.bValue = TRUE THEN
			eTravAct		:= TravActPwrOn;

			IF p_eTravStat = TravActPwrOn AND p_eTravStatus = Done THEN
				eTravAct	:= TravActIdle;

				tyP0936Trav.tyMotionStd.tyBtnPwr.bRtCompl		:= FALSE;
				tyP0936Trav.tyMotionStd.tyBtnPwr.bRtLk			:= FALSE;
			END_IF
		ELSE
			eTravAct		:= TravActPwrOff;

			IF p_eTravStat = TravActPwrOff AND p_eTravStatus = Done THEN
				eTravAct	:= TravActIdle;

				tyP0936Trav.tyMotionStd.tyBtnPwr.bRtCompl		:= FALSE;
				tyP0936Trav.tyMotionStd.tyBtnPwr.bRtLk			:= FALSE;
			END_IF
		END_IF

	ELSIF tyP0936Trav.tyMotionStd.tyBtnOrigin.bRtCompl = TRUE THEN
		tyP0936Trav.tyMotionStd.tyBtnOrigin.bValue				:= TRUE;
		tyP0936Trav.tyMotionStd.tyBtnStop.bValue				:= FALSE;

		tyP0936Trav.tyMotionStd.tyBtnOrigin.bRtLk				:= TRUE;
		tyP0936Trav.tyMotionStd.tyBtnStop.bRtLk					:= FALSE;

		eTravAct		:= TravActHoming;

		IF p_eTravStat = TravActHoming AND p_eTravStatus = Done THEN
			eTravAct	:= TravActIdle;

			tyP0936Trav.tyMotionStd.tyBtnOrigin.bRtCompl		:= FALSE;
			tyP0936Trav.tyMotionStd.tyBtnOrigin.bValue			:= FALSE;
			tyP0936Trav.tyMotionStd.tyBtnStop.bValue			:= TRUE;

			tyP0936Trav.tyMotionStd.tyBtnOrigin.bRtLk			:= FALSE;
			tyP0936Trav.tyMotionStd.tyBtnStop.bRtLk				:= TRUE;
		END_IF

	ELSIF tyP0936Trav.tyMotionStd.tyBtnRst.bRtCompl = TRUE THEN
		tyP0936Trav.tyMotionStd.tyBtnRst.bValue					:= TRUE;
		tyP0936Trav.tyMotionStd.tyBtnRst.bRtLk					:= TRUE;

		eTravAct		:= TravActRstAxisErr;

		IF p_eTravStat = TravActRstAxisErr AND p_eTravStatus = Done THEN
			eTravAct	:= TravActIdle;

			tyP0936Trav.tyMotionStd.tyBtnRst.bRtCompl			:= FALSE;
			tyP0936Trav.tyMotionStd.tyBtnRst.bValue				:= FALSE;
			tyP0936Trav.tyMotionStd.tyBtnRst.bRtLk				:= FALSE;

			fbLmtRstTm.IN			:= FALSE;
		END_IF

	ELSIF tyP0936Trav.tyTrav.tyBtnGoToLaneA.bRtCompl = TRUE THEN
		tyP0936Trav.tyTrav.tyBtnGoToLaneA.bValue				:= TRUE;
		tyP0936Trav.tyMotionStd.tyBtnStop.bValue				:= FALSE;

		tyP0936Trav.tyTrav.tyBtnGoToLaneA.bRtLk					:= TRUE;
		tyP0936Trav.tyMotionStd.tyBtnStop.bRtLk					:= FALSE;

		diMnlTravNomSpd	:= tyP0936Trav.tyMotionStd.tyNumNomSpd.diValue;

		eTravAct		:= TravActGoDPos;

		IF p_eTravStat = TravActGoDPos AND p_eTravStatus = Done THEN
			eTravAct	:= TravActIdle;

			tyP0936Trav.tyTrav.tyBtnGoToLaneA.bRtCompl				:= FALSE;
			tyP0936Trav.tyTrav.tyBtnGoToLaneA.bValue				:= FALSE;
			tyP0936Trav.tyMotionStd.tyBtnStop.bValue				:= TRUE;

			tyP0936Trav.tyTrav.tyBtnGoToLaneA.bRtLk					:= FALSE;
			tyP0936Trav.tyMotionStd.tyBtnStop.bRtLk					:= TRUE;
		END_IF

	ELSIF tyP0936Trav.tyTrav.tyBtnGoToLaneB.bRtCompl = TRUE THEN
		tyP0936Trav.tyTrav.tyBtnGoToLaneB.bValue					:= TRUE;
		tyP0936Trav.tyMotionStd.tyBtnStop.bValue					:= FALSE;

		tyP0936Trav.tyTrav.tyBtnGoToLaneB.bRtLk						:= TRUE;
		tyP0936Trav.tyMotionStd.tyBtnStop.bRtLk						:= FALSE;

		diMnlTravNomSpd	:= tyP0936Trav.tyMotionStd.tyNumNomSpd.diValue;

		eTravAct		:= TravActGoEPos;

		IF p_eTravStat = TravActGoEPos AND p_eTravStatus = Done THEN
			eTravAct	:= TravActIdle;

			tyP0936Trav.tyTrav.tyBtnGoToLaneB.bRtCompl				:= FALSE;
			tyP0936Trav.tyTrav.tyBtnGoToLaneB.bValue				:= FALSE;
			tyP0936Trav.tyMotionStd.tyBtnStop.bValue				:= TRUE;

			tyP0936Trav.tyTrav.tyBtnGoToLaneB.bRtLk					:= FALSE;
			tyP0936Trav.tyMotionStd.tyBtnStop.bRtLk					:= TRUE;
		END_IF

	ELSIF tyP0936Trav.tyTrav.tyBtnGoToMag1.bRtCompl = TRUE THEN
		tyP0936Trav.tyTrav.tyBtnGoToMag1.bValue						:= TRUE;
		tyP0936Trav.tyMotionStd.tyBtnStop.bValue					:= FALSE;

		tyP0936Trav.tyTrav.tyBtnGoToMag1.bRtLk						:= TRUE;
		tyP0936Trav.tyMotionStd.tyBtnStop.bRtLk						:= FALSE;

		diMnlTravNomSpd	:= tyP0936Trav.tyMotionStd.tyNumNomSpd.diValue;

		eTravAct		:= TravActGoAPos;

		IF p_eTravStat = TravActGoAPos AND p_eTravStatus = Done THEN
			eTravAct	:= TravActIdle;

			tyP0936Trav.tyTrav.tyBtnGoToMag1.bRtCompl				:= FALSE;
			tyP0936Trav.tyTrav.tyBtnGoToMag1.bValue					:= FALSE;
			tyP0936Trav.tyMotionStd.tyBtnStop.bValue				:= TRUE;

			tyP0936Trav.tyTrav.tyBtnGoToMag1.bRtLk					:= FALSE;
			tyP0936Trav.tyMotionStd.tyBtnStop.bRtLk					:= TRUE;
		END_IF

	ELSIF tyP0936Trav.tyTrav.tyBtnGoToMag2.bRtCompl = TRUE THEN
		tyP0936Trav.tyTrav.tyBtnGoToMag2.bValue						:= TRUE;
		tyP0936Trav.tyMotionStd.tyBtnStop.bValue					:= FALSE;

		tyP0936Trav.tyTrav.tyBtnGoToMag2.bRtLk						:= TRUE;
		tyP0936Trav.tyMotionStd.tyBtnStop.bRtLk						:= FALSE;

		diMnlTravNomSpd	:= tyP0936Trav.tyMotionStd.tyNumNomSpd.diValue;

		eTravAct		:= TravActGoBPos;

		IF p_eTravStat = TravActGoBPos AND p_eTravStatus = Done THEN
			eTravAct	:= TravActIdle;

			tyP0936Trav.tyTrav.tyBtnGoToMag2.bRtCompl				:= FALSE;
			tyP0936Trav.tyTrav.tyBtnGoToMag2.bValue					:= FALSE;
			tyP0936Trav.tyMotionStd.tyBtnStop.bValue				:= TRUE;

			tyP0936Trav.tyTrav.tyBtnGoToMag2.bRtLk					:= FALSE;
			tyP0936Trav.tyMotionStd.tyBtnStop.bRtLk					:= TRUE;
		END_IF

	ELSIF tyP0936Trav.tyTrav.tyBtnGoToMag3.bRtCompl = TRUE THEN
		tyP0936Trav.tyTrav.tyBtnGoToMag3.bValue						:= TRUE;
		tyP0936Trav.tyMotionStd.tyBtnStop.bValue					:= FALSE;

		tyP0936Trav.tyTrav.tyBtnGoToMag3.bRtLk						:= TRUE;
		tyP0936Trav.tyMotionStd.tyBtnStop.bRtLk						:= FALSE;

		diMnlTravNomSpd	:= tyP0936Trav.tyMotionStd.tyNumNomSpd.diValue;

		eTravAct		:= TravActGoCPos;

		IF p_eTravStat = TravActGoCPos AND p_eTravStatus = Done THEN
			eTravAct	:= TravActIdle;

			tyP0936Trav.tyTrav.tyBtnGoToMag3.bRtCompl				:= FALSE;
			tyP0936Trav.tyTrav.tyBtnGoToMag3.bValue					:= FALSE;
			tyP0936Trav.tyMotionStd.tyBtnStop.bValue				:= TRUE;

			tyP0936Trav.tyTrav.tyBtnGoToMag3.bRtLk					:= FALSE;
			tyP0936Trav.tyMotionStd.tyBtnStop.bRtLk					:= TRUE;
		END_IF

	ELSIF tyP0936Trav.tyTrav.tyBtnGoToMag4.bRtCompl = TRUE THEN
		tyP0936Trav.tyTrav.tyBtnGoToMag4.bValue						:= TRUE;
		tyP0936Trav.tyMotionStd.tyBtnStop.bValue					:= FALSE;

		tyP0936Trav.tyTrav.tyBtnGoToMag4.bRtLk						:= TRUE;
		tyP0936Trav.tyMotionStd.tyBtnStop.bRtLk						:= FALSE;

		diMnlTravNomSpd	:= tyP0936Trav.tyMotionStd.tyNumNomSpd.diValue;

		eTravAct		:= TravActGoGPos;

		IF p_eTravStat = TravActGoGPos AND p_eTravStatus = Done THEN
			eTravAct	:= TravActIdle;

			tyP0936Trav.tyTrav.tyBtnGoToMag4.bRtCompl				:= FALSE;
			tyP0936Trav.tyTrav.tyBtnGoToMag4.bValue					:= FALSE;
			tyP0936Trav.tyMotionStd.tyBtnStop.bValue				:= TRUE;

			tyP0936Trav.tyTrav.tyBtnGoToMag4.bRtLk					:= FALSE;
			tyP0936Trav.tyMotionStd.tyBtnStop.bRtLk					:= TRUE;
		END_IF

	ELSIF tyP0936Trav.tyMotionStd.tyBtnMovAbs.bRtCompl = TRUE THEN
		tyP0936Trav.tyMotionStd.tyBtnMovAbs.bValue				:= TRUE;
		tyP0936Trav.tyMotionStd.tyBtnStop.bValue				:= FALSE;

		tyP0936Trav.tyMotionStd.tyBtnMovAbs.bRtLk				:= TRUE;
		tyP0936Trav.tyMotionStd.tyBtnStop.bRtLk					:= FALSE;

		diMnlTravTargetPos	:= tyP0936Trav.tyMotionStd.tyNumTargetPos.diValue;
		diMnlTravNomSpd		:= tyP0936Trav.tyMotionStd.tyNumNomSpd.diValue;

		eTravAct		:= TravActMovAbs;

		IF p_eTravStat = TravActMovAbs AND p_eTravStatus = Done THEN
			eTravAct	:= TravActIdle;

			tyP0936Trav.tyMotionStd.tyBtnMovAbs.bRtCompl		:= FALSE;
			tyP0936Trav.tyMotionStd.tyBtnMovAbs.bValue			:= FALSE;
			tyP0936Trav.tyMotionStd.tyBtnStop.bValue			:= TRUE;

			tyP0936Trav.tyMotionStd.tyBtnMovAbs.bRtLk			:= FALSE;
			tyP0936Trav.tyMotionStd.tyBtnStop.bRtLk				:= TRUE;
		END_IF

	ELSIF tyP0936Trav.tyMotionStd.tyBtnMovRel.bRtCompl = TRUE THEN
		tyP0936Trav.tyMotionStd.tyBtnMovRel.bValue				:= TRUE;
		tyP0936Trav.tyMotionStd.tyBtnStop.bValue				:= FALSE;

		tyP0936Trav.tyMotionStd.tyBtnMovRel.bRtLk				:= TRUE;
		tyP0936Trav.tyMotionStd.tyBtnStop.bRtLk					:= FALSE;

		diMnlTravStepSize	:= tyP0936Trav.tyMotionStd.tyNumStepSize.diValue;
		diMnlTravNomSpd		:= tyP0936Trav.tyMotionStd.tyNumNomSpd.diValue;

		eTravAct		:= TravActMovRel;

		IF p_eTravStat = TravActMovRel AND p_eTravStatus = Done THEN
			eTravAct	:= TravActIdle;

			tyP0936Trav.tyMotionStd.tyBtnMovRel.bRtCompl		:= FALSE;
			tyP0936Trav.tyMotionStd.tyBtnMovRel.bValue			:= FALSE;
			tyP0936Trav.tyMotionStd.tyBtnStop.bValue			:= TRUE;

			tyP0936Trav.tyMotionStd.tyBtnMovRel.bRtLk			:= FALSE;
			tyP0936Trav.tyMotionStd.tyBtnStop.bRtLk				:= TRUE;
		END_IF

	ELSIF (tyP0936Trav.tyMotionStd.tyBtnJogRear.bValue = TRUE) AND (fbJogSlowToFastDlyTm.Q = FALSE) AND (bJogSlow = FALSE) THEN
		tyP0936Trav.tyMotionStd.tyBtnStop.bValue				:= FALSE;
		tyP0936Trav.tyMotionStd.tyBtnStop.bRtLk					:= FALSE;

		fbJogSlowToFastDlyTm.IN		:= TRUE;

		diMnlTravJogSpd	:= tyP0936Trav.tyMotionStd.tyNumSlwSpd.diValue;

		eTravAct		:= TravActJogRear;

		IF p_eTravStat = TravActJogRear AND p_eTravStatus = Done THEN
			eTravAct	:= TravActIdle;
			bJogSlow				:= TRUE;
		ELSIF p_eTravStatus = Error THEN
			fbJogSlowToFastDlyTm.IN	:= FALSE;
			bJogSlow				:= TRUE;
		END_IF

	ELSIF (tyP0936Trav.tyMotionStd.tyBtnJogRear.bValue = TRUE) AND (fbJogSlowToFastDlyTm.Q = TRUE) AND (bJogFast = FALSE) THEN
		tyP0936Trav.tyMotionStd.tyBtnStop.bValue					:= FALSE;
		tyP0936Trav.tyMotionStd.tyBtnStop.bRtLk						:= FALSE;

		fbJogSlowToFastDlyTm.IN		:= TRUE;

		diMnlTravJogSpd	:= tyP0936Trav.tyMotionStd.tyNumNomSpd.diValue;

		eTravAct		:= TravActJogRear;

		IF p_eTravStat = TravActJogRear AND p_eTravStatus = Done THEN
			eTravAct	:= TravActIdle;
			bJogFast				:= TRUE;
		ELSIF p_eTravStatus = Error THEN
			fbJogSlowToFastDlyTm.IN	:= FALSE;
			bJogFast				:= TRUE;
		END_IF

	ELSIF (tyP0936Trav.tyMotionStd.tyBtnJogFront.bValue = TRUE) AND (fbJogSlowToFastDlyTm.Q = FALSE) AND (bJogSlow = FALSE) THEN
		tyP0936Trav.tyMotionStd.tyBtnStop.bValue				:= FALSE;
		tyP0936Trav.tyMotionStd.tyBtnStop.bRtLk					:= FALSE;

		fbJogSlowToFastDlyTm.IN		:= TRUE;

		diMnlTravJogSpd	:= tyP0936Trav.tyMotionStd.tyNumSlwSpd.diValue;

		eTravAct		:= TravActJogFront;

		IF p_eTravStat = TravActJogFront AND p_eTravStatus = Done THEN
			eTravAct	:= TravActIdle;
			bJogSlow				:= TRUE;
		ELSIF p_eTravStatus = Error THEN
			fbJogSlowToFastDlyTm.IN	:= FALSE;
			bJogSlow				:= TRUE;
		END_IF

	ELSIF (tyP0936Trav.tyMotionStd.tyBtnJogFront.bValue = TRUE) AND (fbJogSlowToFastDlyTm.Q = TRUE) AND (bJogFast = FALSE) THEN

		tyP0936Trav.tyMotionStd.tyBtnStop.bValue				:= FALSE;
		tyP0936Trav.tyMotionStd.tyBtnStop.bRtLk					:= FALSE;

		fbJogSlowToFastDlyTm.IN		:= TRUE;

		diMnlTravJogSpd	:= tyP0936Trav.tyMotionStd.tyNumNomSpd.diValue;

		eTravAct		:= TravActJogFront;

		IF p_eTravStat = TravActJogFront AND p_eTravStatus = Done THEN
			eTravAct	:= TravActIdle;
			bJogFast	:= TRUE;
		ELSIF p_eTravStatus = Error THEN
			fbJogSlowToFastDlyTm.IN	:= FALSE;
			bJogFast				:= TRUE;
		END_IF
	END_IF

	//Shutter Control
	IF tyP0936Trav.tyInOutletShutterFB.tyBtnOpen.bRtCompl = TRUE THEN
		tyP0936Trav.tyInOutletShutterFB.tyBtnOpen.bRtCompl	:= FALSE;

		tyP0936Trav.tyInOutletShutterFB.tyBtnOpen.bValue	:= TRUE;
		tyP0936Trav.tyInOutletShutterFB.tyBtnClose.bValue	:= FALSE;

	ELSIF tyP0936Trav.tyInOutletShutterFB.tyBtnClose.bRtCompl = TRUE THEN
		tyP0936Trav.tyInOutletShutterFB.tyBtnClose.bRtCompl	:= FALSE;

		tyP0936Trav.tyInOutletShutterFB.tyBtnClose.bValue	:= TRUE;
		tyP0936Trav.tyInOutletShutterFB.tyBtnOpen.bValue	:= FALSE;
	END_IF

	IF tyP0936Trav.tyInOutletShutterFB.tyBtnOpen.bValue = TRUE THEN
		eInShutterAct	:= PneuActRet;
		eOutShutterAct	:= PneuActRet;

		IF (p_eInShutterStat = PneuActRet AND p_eInShutterStatus = Done)
			AND (p_eOutShutterStat = PneuActRet AND p_eOutShutterStatus = Done)
			THEN
			eInShutterAct	:= PneuActIdle;
			eOutShutterAct	:= PneuActIdle;
			tyP0936Trav.tyInOutletShutterFB.tyBtnOpen.bValue	:= FALSE;
		ELSIF p_eInShutterStatus = Error OR p_eOutShutterStatus = Error THEN
			tyP0936Trav.tyInOutletShutterFB.tyBtnOpen.bValue	:= FALSE;
		END_IF

	ELSIF tyP0936Trav.tyInOutletShutterFB.tyBtnClose.bValue = TRUE THEN
		eInShutterAct	:= PneuActExt;
		eOutShutterAct	:= PneuActExt;
		IF (p_eInShutterStat = PneuActExt AND p_eInShutterStatus = Done)
			AND (p_eOutShutterStat = PneuActExt AND p_eOutShutterStatus = Done)
			THEN
			eInShutterAct	:= PneuActIdle;
			eOutShutterAct	:= PneuActIdle;
			tyP0936Trav.tyInOutletShutterFB.tyBtnClose.bValue := FALSE;
		ELSIF p_eInShutterStatus = Error OR p_eOutShutterStatus = Error THEN
			tyP0936Trav.tyInOutletShutterFB.tyBtnClose.bValue := FALSE;
		END_IF
	END_IF

END_ACTION
```

#### Act_OptP0936FullMask.st
```iecst
ACTION Act_OptP0936FullMask:

	IF eCurrPage = UIP0936Trav THEN

		IF p_tyDI.bEStopSig = FALSE THEN
			p_tyC0002FullMask ACCESS ADR(tyP0936Trav.tyFullMaskEStop);

		ELSIF p_tyDI.bCoverSWSig = FALSE THEN
			p_tyC0002FullMask ACCESS ADR(tyP0936Trav.tyFullMaskCWSig);

		ELSIF p_tyDI.bSafetyRlySig = FALSE THEN
			p_tyC0002FullMask ACCESS ADR(tyP0936Trav.tyFullMaskSafetyRly);

		ELSIF p_tyDI.bConvLftSen THEN
			p_tyC0002FullMask ACCESS ADR(tyP0936Trav.tyFullMaskLftSenInterrupt);

		ELSIF p_tyDI.bConvRgtSen THEN
			p_tyC0002FullMask ACCESS ADR(tyP0936Trav.tyFullMaskRgtSenInterrupt);

		ELSIF p_tyDI.bPullerRetRS = FALSE OR p_tyDI.bPullerRotHmRS = FALSE THEN
			p_tyC0002FullMask ACCESS ADR(tyP0936Trav.tyFullMaskPullInterrupt);

		ELSIF p_tyNtParamCurr.bProjInletShutPrep AND (p_tyDI.bInShutterCloseRS = FALSE
			OR (p_tyDI.bInShutterCloseRS2 = FALSE AND p_tyNtParamCurr.tyDISettings.diInShutterCloseRS2 > 0)
			OR (p_tyDI.bInShutterCloseRS3 = FALSE AND p_tyNtParamCurr.tyDISettings.diInShutterCloseRS3 > 0)) THEN
			IF p_tyNtParamCurr.bProjCurtainSenPrep THEN
				IF p_tyDI.bInShutterCloseRS = FALSE OR p_tyDI.bInShutterCloseRS2 = FALSE OR p_tyDI.bInShutterCloseRS3 = FALSE THEN
					p_tyC0002FullMask ACCESS ADR(tyP0936Trav.tyFullMaskInShutOpnInterrupt);
				END_IF
			ELSE
				IF p_tyDI.bInShutterCloseRS = FALSE THEN
					p_tyC0002FullMask ACCESS ADR(tyP0936Trav.tyFullMaskInShutOpnInterrupt);
				END_IF
			END_IF

	//	ELSIF p_tyNtParamCurr.bProjOutletShutPrep AND p_tyDI.bOutShutterCloseRS = FALSE AND p_McParamOutShutterDis = FALSE THEN
		ELSIF p_tyNtParamCurr.bProjOutletShutPrep AND p_tyDI.bOutShutterCloseRS = FALSE THEN
			p_tyC0002FullMask ACCESS ADR(tyP0936Trav.tyFullMaskOutShutOpnInterrupt);

		ELSE
			p_tyC0002FullMask ACCESS ADR(tyP0936Trav.tyFullMaskHide);

		END_IF

	END_IF

END_ACTION
```

#### Act_OptP0936Mask.st
```iecst
ACTION Act_OptP0936Mask:

	// Interlock Power
	IF p_bTravAxisErr = TRUE AND p_bTravPwrOn = FALSE THEN
		fUIInRtStatOff(ADR(tyP0936Trav.tyMotionStd.tyBtnPwr.uiMaskRtStat));
		tyP0936Trav.tyMotionStd.tyBtnPwr.bValue		:= FALSE;
	ELSE
		fUIInRtStatHide(ADR(tyP0936Trav.tyMotionStd.tyBtnPwr.uiMaskRtStat));
	END_IF

	// Interlock Others Move
	IF p_bTravAxisErr = TRUE OR p_bTravPwrOn = FALSE THEN
		fUIInRtStatOff(ADR(tyP0936Trav.tyMotionStd.tyBtnOrigin.uiMaskRtStat));
		fUIInRtStatOff(ADR(tyP0936Trav.tyMotionStd.tyBtnMovRel.uiMaskRtStat));
		fUIInRtStatOff(ADR(tyP0936Trav.tyMotionStd.tyBtnJogFront.uiMaskRtStat));
		fUIInRtStatOff(ADR(tyP0936Trav.tyMotionStd.tyBtnJogRear.uiMaskRtStat));
	ELSE
		fUIInRtStatHide(ADR(tyP0936Trav.tyMotionStd.tyBtnOrigin.uiMaskRtStat));
		fUIInRtStatHide(ADR(tyP0936Trav.tyMotionStd.tyBtnMovRel.uiMaskRtStat));
		fUIInRtStatHide(ADR(tyP0936Trav.tyMotionStd.tyBtnJogFront.uiMaskRtStat));
		fUIInRtStatHide(ADR(tyP0936Trav.tyMotionStd.tyBtnJogRear.uiMaskRtStat));
	END_IF

	// Interlock Move Absolute
	IF p_bTravAxisErr = TRUE OR p_bTravPwrOn = FALSE OR p_bTravIsHomed = FALSE THEN
		fUIInRtStatOff(ADR(tyP0936Trav.tyTrav.tyBtnGoToLaneA.uiMaskRtStat));
		fUIInRtStatOff(ADR(tyP0936Trav.tyTrav.tyBtnGoToLaneB.uiMaskRtStat));
		fUIInRtStatOff(ADR(tyP0936Trav.tyTrav.tyBtnGoToMag1.uiMaskRtStat));
		fUIInRtStatOff(ADR(tyP0936Trav.tyTrav.tyBtnGoToMag2.uiMaskRtStat));
		fUIInRtStatOff(ADR(tyP0936Trav.tyTrav.tyBtnGoToMag3.uiMaskRtStat));
		fUIInRtStatOff(ADR(tyP0936Trav.tyTrav.tyBtnGoToMag4.uiMaskRtStat));
		fUIInRtStatOff(ADR(tyP0936Trav.tyMotionStd.tyBtnMovAbs.uiMaskRtStat));
	ELSE
		fUIInRtStatHide(ADR(tyP0936Trav.tyTrav.tyBtnGoToLaneA.uiMaskRtStat));
		fUIInRtStatHide(ADR(tyP0936Trav.tyTrav.tyBtnGoToLaneB.uiMaskRtStat));
		fUIInRtStatHide(ADR(tyP0936Trav.tyTrav.tyBtnGoToMag1.uiMaskRtStat));
		fUIInRtStatHide(ADR(tyP0936Trav.tyTrav.tyBtnGoToMag2.uiMaskRtStat));
		fUIInRtStatHide(ADR(tyP0936Trav.tyTrav.tyBtnGoToMag3.uiMaskRtStat));
		fUIInRtStatHide(ADR(tyP0936Trav.tyTrav.tyBtnGoToMag4.uiMaskRtStat));
		fUIInRtStatHide(ADR(tyP0936Trav.tyMotionStd.tyBtnMovAbs.uiMaskRtStat));
	END_IF

	//Interlock Limit Sensor
	IF tyP0936Trav.tyMotionStd.tyBtnRearLmtSen.bValue = TRUE THEN
		fUIInRtStatOff(ADR(tyP0936Trav.tyMotionStd.tyBtnJogRear.uiMaskRtStat));
	END_IF

	IF tyP0936Trav.tyMotionStd.tyBtnFrontLmtSen.bValue = TRUE THEN
		fUIInRtStatOff(ADR(tyP0936Trav.tyMotionStd.tyBtnJogFront.uiMaskRtStat));
	END_IF

	// Interlock When Moving
	IF tyP0936Trav.tyMotionStd.tyBtnOrigin.bRtCompl = TRUE THEN
		fUIInRtStatOff(ADR(tyP0936Trav.tyMotionStd.tyBtnMovAbs.uiMaskRtStat));
		fUIInRtStatOff(ADR(tyP0936Trav.tyMotionStd.tyBtnMovRel.uiMaskRtStat));
		fUIInRtStatOff(ADR(tyP0936Trav.tyMotionStd.tyBtnJogFront.uiMaskRtStat));
		fUIInRtStatOff(ADR(tyP0936Trav.tyMotionStd.tyBtnJogRear.uiMaskRtStat));
		fUIInRtStatOff(ADR(tyP0936Trav.tyTrav.tyBtnGoToLaneA.uiMaskRtStat));
		fUIInRtStatOff(ADR(tyP0936Trav.tyTrav.tyBtnGoToLaneB.uiMaskRtStat));
		fUIInRtStatOff(ADR(tyP0936Trav.tyTrav.tyBtnGoToMag1.uiMaskRtStat));
		fUIInRtStatOff(ADR(tyP0936Trav.tyTrav.tyBtnGoToMag2.uiMaskRtStat));
		fUIInRtStatOff(ADR(tyP0936Trav.tyTrav.tyBtnGoToMag3.uiMaskRtStat));
		fUIInRtStatOff(ADR(tyP0936Trav.tyTrav.tyBtnGoToMag4.uiMaskRtStat));

	ELSIF tyP0936Trav.tyMotionStd.tyBtnMovAbs.bRtCompl = TRUE THEN
		fUIInRtStatOff(ADR(tyP0936Trav.tyMotionStd.tyBtnOrigin.uiMaskRtStat));
		fUIInRtStatOff(ADR(tyP0936Trav.tyMotionStd.tyBtnMovRel.uiMaskRtStat));
		fUIInRtStatOff(ADR(tyP0936Trav.tyMotionStd.tyBtnJogFront.uiMaskRtStat));
		fUIInRtStatOff(ADR(tyP0936Trav.tyMotionStd.tyBtnJogRear.uiMaskRtStat));
		fUIInRtStatOff(ADR(tyP0936Trav.tyTrav.tyBtnGoToLaneA.uiMaskRtStat));
		fUIInRtStatOff(ADR(tyP0936Trav.tyTrav.tyBtnGoToLaneB.uiMaskRtStat));
		fUIInRtStatOff(ADR(tyP0936Trav.tyTrav.tyBtnGoToMag1.uiMaskRtStat));
		fUIInRtStatOff(ADR(tyP0936Trav.tyTrav.tyBtnGoToMag2.uiMaskRtStat));
		fUIInRtStatOff(ADR(tyP0936Trav.tyTrav.tyBtnGoToMag3.uiMaskRtStat));
		fUIInRtStatOff(ADR(tyP0936Trav.tyTrav.tyBtnGoToMag4.uiMaskRtStat));

	ELSIF tyP0936Trav.tyMotionStd.tyBtnMovRel.bRtCompl = TRUE THEN
		fUIInRtStatOff(ADR(tyP0936Trav.tyMotionStd.tyBtnOrigin.uiMaskRtStat));
		fUIInRtStatOff(ADR(tyP0936Trav.tyMotionStd.tyBtnMovAbs.uiMaskRtStat));
		fUIInRtStatOff(ADR(tyP0936Trav.tyMotionStd.tyBtnJogFront.uiMaskRtStat));
		fUIInRtStatOff(ADR(tyP0936Trav.tyMotionStd.tyBtnJogRear.uiMaskRtStat));
		fUIInRtStatOff(ADR(tyP0936Trav.tyTrav.tyBtnGoToLaneA.uiMaskRtStat));
		fUIInRtStatOff(ADR(tyP0936Trav.tyTrav.tyBtnGoToLaneB.uiMaskRtStat));
		fUIInRtStatOff(ADR(tyP0936Trav.tyTrav.tyBtnGoToMag1.uiMaskRtStat));
		fUIInRtStatOff(ADR(tyP0936Trav.tyTrav.tyBtnGoToMag2.uiMaskRtStat));
		fUIInRtStatOff(ADR(tyP0936Trav.tyTrav.tyBtnGoToMag3.uiMaskRtStat));
		fUIInRtStatOff(ADR(tyP0936Trav.tyTrav.tyBtnGoToMag4.uiMaskRtStat));

	ELSIF tyP0936Trav.tyMotionStd.tyBtnJogRear.bRtCompl = TRUE OR tyP0936Trav.tyMotionStd.tyBtnJogRear.bValue = TRUE THEN
		fUIInRtStatOff(ADR(tyP0936Trav.tyMotionStd.tyBtnOrigin.uiMaskRtStat));
		fUIInRtStatOff(ADR(tyP0936Trav.tyMotionStd.tyBtnMovAbs.uiMaskRtStat));
		fUIInRtStatOff(ADR(tyP0936Trav.tyMotionStd.tyBtnMovRel.uiMaskRtStat));
		fUIInRtStatOff(ADR(tyP0936Trav.tyMotionStd.tyBtnJogFront.uiMaskRtStat));
		fUIInRtStatOff(ADR(tyP0936Trav.tyTrav.tyBtnGoToLaneA.uiMaskRtStat));
		fUIInRtStatOff(ADR(tyP0936Trav.tyTrav.tyBtnGoToLaneB.uiMaskRtStat));
		fUIInRtStatOff(ADR(tyP0936Trav.tyTrav.tyBtnGoToMag1.uiMaskRtStat));
		fUIInRtStatOff(ADR(tyP0936Trav.tyTrav.tyBtnGoToMag2.uiMaskRtStat));
		fUIInRtStatOff(ADR(tyP0936Trav.tyTrav.tyBtnGoToMag3.uiMaskRtStat));
		fUIInRtStatOff(ADR(tyP0936Trav.tyTrav.tyBtnGoToMag4.uiMaskRtStat));

	ELSIF tyP0936Trav.tyMotionStd.tyBtnJogFront.bRtCompl = TRUE OR tyP0936Trav.tyMotionStd.tyBtnJogFront.bValue = TRUE THEN
		fUIInRtStatOff(ADR(tyP0936Trav.tyMotionStd.tyBtnOrigin.uiMaskRtStat));
		fUIInRtStatOff(ADR(tyP0936Trav.tyMotionStd.tyBtnMovAbs.uiMaskRtStat));
		fUIInRtStatOff(ADR(tyP0936Trav.tyMotionStd.tyBtnMovRel.uiMaskRtStat));
		fUIInRtStatOff(ADR(tyP0936Trav.tyMotionStd.tyBtnJogRear.uiMaskRtStat));
		fUIInRtStatOff(ADR(tyP0936Trav.tyTrav.tyBtnGoToLaneA.uiMaskRtStat));
		fUIInRtStatOff(ADR(tyP0936Trav.tyTrav.tyBtnGoToLaneB.uiMaskRtStat));
		fUIInRtStatOff(ADR(tyP0936Trav.tyTrav.tyBtnGoToMag1.uiMaskRtStat));
		fUIInRtStatOff(ADR(tyP0936Trav.tyTrav.tyBtnGoToMag2.uiMaskRtStat));
		fUIInRtStatOff(ADR(tyP0936Trav.tyTrav.tyBtnGoToMag3.uiMaskRtStat));
		fUIInRtStatOff(ADR(tyP0936Trav.tyTrav.tyBtnGoToMag4.uiMaskRtStat));

	ELSIF tyP0936Trav.tyTrav.tyBtnGoToLaneA.bRtCompl = TRUE THEN
		fUIInRtStatOff(ADR(tyP0936Trav.tyMotionStd.tyBtnOrigin.uiMaskRtStat));
		fUIInRtStatOff(ADR(tyP0936Trav.tyMotionStd.tyBtnMovAbs.uiMaskRtStat));
		fUIInRtStatOff(ADR(tyP0936Trav.tyMotionStd.tyBtnMovRel.uiMaskRtStat));
		fUIInRtStatOff(ADR(tyP0936Trav.tyMotionStd.tyBtnJogFront.uiMaskRtStat));
		fUIInRtStatOff(ADR(tyP0936Trav.tyMotionStd.tyBtnJogRear.uiMaskRtStat));
		fUIInRtStatOff(ADR(tyP0936Trav.tyTrav.tyBtnGoToLaneB.uiMaskRtStat));
		fUIInRtStatOff(ADR(tyP0936Trav.tyTrav.tyBtnGoToMag1.uiMaskRtStat));
		fUIInRtStatOff(ADR(tyP0936Trav.tyTrav.tyBtnGoToMag2.uiMaskRtStat));
		fUIInRtStatOff(ADR(tyP0936Trav.tyTrav.tyBtnGoToMag3.uiMaskRtStat));
		fUIInRtStatOff(ADR(tyP0936Trav.tyTrav.tyBtnGoToMag4.uiMaskRtStat));

	ELSIF tyP0936Trav.tyTrav.tyBtnGoToLaneB.bRtCompl = TRUE THEN
		fUIInRtStatOff(ADR(tyP0936Trav.tyMotionStd.tyBtnOrigin.uiMaskRtStat));
		fUIInRtStatOff(ADR(tyP0936Trav.tyMotionStd.tyBtnMovAbs.uiMaskRtStat));
		fUIInRtStatOff(ADR(tyP0936Trav.tyMotionStd.tyBtnMovRel.uiMaskRtStat));
		fUIInRtStatOff(ADR(tyP0936Trav.tyMotionStd.tyBtnJogFront.uiMaskRtStat));
		fUIInRtStatOff(ADR(tyP0936Trav.tyMotionStd.tyBtnJogRear.uiMaskRtStat));
		fUIInRtStatOff(ADR(tyP0936Trav.tyTrav.tyBtnGoToLaneA.uiMaskRtStat));
		fUIInRtStatOff(ADR(tyP0936Trav.tyTrav.tyBtnGoToMag1.uiMaskRtStat));
		fUIInRtStatOff(ADR(tyP0936Trav.tyTrav.tyBtnGoToMag2.uiMaskRtStat));
		fUIInRtStatOff(ADR(tyP0936Trav.tyTrav.tyBtnGoToMag3.uiMaskRtStat));
		fUIInRtStatOff(ADR(tyP0936Trav.tyTrav.tyBtnGoToMag4.uiMaskRtStat));

	ELSIF tyP0936Trav.tyTrav.tyBtnGoToMag1.bRtCompl = TRUE THEN
		fUIInRtStatOff(ADR(tyP0936Trav.tyMotionStd.tyBtnOrigin.uiMaskRtStat));
		fUIInRtStatOff(ADR(tyP0936Trav.tyMotionStd.tyBtnMovAbs.uiMaskRtStat));
		fUIInRtStatOff(ADR(tyP0936Trav.tyMotionStd.tyBtnMovRel.uiMaskRtStat));
		fUIInRtStatOff(ADR(tyP0936Trav.tyMotionStd.tyBtnJogFront.uiMaskRtStat));
		fUIInRtStatOff(ADR(tyP0936Trav.tyMotionStd.tyBtnJogRear.uiMaskRtStat));
		fUIInRtStatOff(ADR(tyP0936Trav.tyTrav.tyBtnGoToLaneA.uiMaskRtStat));
		fUIInRtStatOff(ADR(tyP0936Trav.tyTrav.tyBtnGoToLaneB.uiMaskRtStat));
		fUIInRtStatOff(ADR(tyP0936Trav.tyTrav.tyBtnGoToMag2.uiMaskRtStat));
		fUIInRtStatOff(ADR(tyP0936Trav.tyTrav.tyBtnGoToMag3.uiMaskRtStat));
		fUIInRtStatOff(ADR(tyP0936Trav.tyTrav.tyBtnGoToMag4.uiMaskRtStat));

	ELSIF tyP0936Trav.tyTrav.tyBtnGoToMag2.bRtCompl = TRUE THEN
		fUIInRtStatOff(ADR(tyP0936Trav.tyMotionStd.tyBtnOrigin.uiMaskRtStat));
		fUIInRtStatOff(ADR(tyP0936Trav.tyMotionStd.tyBtnMovAbs.uiMaskRtStat));
		fUIInRtStatOff(ADR(tyP0936Trav.tyMotionStd.tyBtnMovRel.uiMaskRtStat));
		fUIInRtStatOff(ADR(tyP0936Trav.tyMotionStd.tyBtnJogFront.uiMaskRtStat));
		fUIInRtStatOff(ADR(tyP0936Trav.tyMotionStd.tyBtnJogRear.uiMaskRtStat));
		fUIInRtStatOff(ADR(tyP0936Trav.tyTrav.tyBtnGoToLaneA.uiMaskRtStat));
		fUIInRtStatOff(ADR(tyP0936Trav.tyTrav.tyBtnGoToLaneB.uiMaskRtStat));
		fUIInRtStatOff(ADR(tyP0936Trav.tyTrav.tyBtnGoToMag1.uiMaskRtStat));
		fUIInRtStatOff(ADR(tyP0936Trav.tyTrav.tyBtnGoToMag3.uiMaskRtStat));
		fUIInRtStatOff(ADR(tyP0936Trav.tyTrav.tyBtnGoToMag4.uiMaskRtStat));

	ELSIF tyP0936Trav.tyTrav.tyBtnGoToMag3.bRtCompl = TRUE THEN
		fUIInRtStatOff(ADR(tyP0936Trav.tyMotionStd.tyBtnOrigin.uiMaskRtStat));
		fUIInRtStatOff(ADR(tyP0936Trav.tyMotionStd.tyBtnMovAbs.uiMaskRtStat));
		fUIInRtStatOff(ADR(tyP0936Trav.tyMotionStd.tyBtnMovRel.uiMaskRtStat));
		fUIInRtStatOff(ADR(tyP0936Trav.tyMotionStd.tyBtnJogFront.uiMaskRtStat));
		fUIInRtStatOff(ADR(tyP0936Trav.tyMotionStd.tyBtnJogRear.uiMaskRtStat));
		fUIInRtStatOff(ADR(tyP0936Trav.tyTrav.tyBtnGoToLaneA.uiMaskRtStat));
		fUIInRtStatOff(ADR(tyP0936Trav.tyTrav.tyBtnGoToLaneB.uiMaskRtStat));
		fUIInRtStatOff(ADR(tyP0936Trav.tyTrav.tyBtnGoToMag1.uiMaskRtStat));
		fUIInRtStatOff(ADR(tyP0936Trav.tyTrav.tyBtnGoToMag2.uiMaskRtStat));
		fUIInRtStatOff(ADR(tyP0936Trav.tyTrav.tyBtnGoToMag4.uiMaskRtStat));

	ELSIF tyP0936Trav.tyTrav.tyBtnGoToMag4.bRtCompl = TRUE THEN
		fUIInRtStatOff(ADR(tyP0936Trav.tyMotionStd.tyBtnOrigin.uiMaskRtStat));
		fUIInRtStatOff(ADR(tyP0936Trav.tyMotionStd.tyBtnMovAbs.uiMaskRtStat));
		fUIInRtStatOff(ADR(tyP0936Trav.tyMotionStd.tyBtnMovRel.uiMaskRtStat));
		fUIInRtStatOff(ADR(tyP0936Trav.tyMotionStd.tyBtnJogFront.uiMaskRtStat));
		fUIInRtStatOff(ADR(tyP0936Trav.tyMotionStd.tyBtnJogRear.uiMaskRtStat));
		fUIInRtStatOff(ADR(tyP0936Trav.tyTrav.tyBtnGoToLaneA.uiMaskRtStat));
		fUIInRtStatOff(ADR(tyP0936Trav.tyTrav.tyBtnGoToLaneB.uiMaskRtStat));
		fUIInRtStatOff(ADR(tyP0936Trav.tyTrav.tyBtnGoToMag1.uiMaskRtStat));
		fUIInRtStatOff(ADR(tyP0936Trav.tyTrav.tyBtnGoToMag2.uiMaskRtStat));
		fUIInRtStatOff(ADR(tyP0936Trav.tyTrav.tyBtnGoToMag3.uiMaskRtStat));
	END_IF

	//Axis Error
	IF tyP0936Trav.tyMotionStd.tyBtnPwr.bRtCompl = TRUE THEN
		fUIInRtStatOff(ADR(tyP0936Trav.tyMotionStd.tyBtnRst.uiMaskRtStat));
	ELSE
		fUIInRtStatHide(ADR(tyP0936Trav.tyMotionStd.tyBtnRst.uiMaskRtStat));
	END_IF

END_ACTION
```

#### Act_OptP0936RstMnl.st
```iecst
ACTION Act_OptP0936RstMnl:

	IF EDGEPOS((bManualMod = FALSE) OR (p_eTravStatus = Error)) THEN

		eTravAct	:= TravActIdle;

		bJogSlow				:= FALSE;
		bJogFast				:= FALSE;
		fbJogSlowToFastDlyTm.IN	:= FALSE;

		tyP0936Trav.tyTrav.tyBtnGoToLaneA.bRtCompl				:= FALSE;
		tyP0936Trav.tyTrav.tyBtnGoToLaneA.bValue				:= FALSE;
		tyP0936Trav.tyTrav.tyBtnGoToLaneA.bRtLk					:= FALSE;
		tyP0936Trav.tyTrav.tyBtnGoToLaneA.uiMaskRtStat.0		:= FALSE;

		tyP0936Trav.tyTrav.tyBtnGoToLaneB.bRtCompl				:= FALSE;
		tyP0936Trav.tyTrav.tyBtnGoToLaneB.bValue				:= FALSE;
		tyP0936Trav.tyTrav.tyBtnGoToLaneB.bRtLk					:= FALSE;
		tyP0936Trav.tyTrav.tyBtnGoToLaneB.uiMaskRtStat.0		:= FALSE;

		tyP0936Trav.tyTrav.tyBtnGoToMag1.bRtCompl				:= FALSE;
		tyP0936Trav.tyTrav.tyBtnGoToMag1.bValue					:= FALSE;
		tyP0936Trav.tyTrav.tyBtnGoToMag1.bRtLk					:= FALSE;
		tyP0936Trav.tyTrav.tyBtnGoToMag1.uiMaskRtStat.0			:= FALSE;

		tyP0936Trav.tyTrav.tyBtnGoToMag2.bRtCompl				:= FALSE;
		tyP0936Trav.tyTrav.tyBtnGoToMag2.bValue					:= FALSE;
		tyP0936Trav.tyTrav.tyBtnGoToMag2.bRtLk					:= FALSE;
		tyP0936Trav.tyTrav.tyBtnGoToMag2.uiMaskRtStat.0			:= FALSE;

		tyP0936Trav.tyTrav.tyBtnGoToMag3.bRtCompl				:= FALSE;
		tyP0936Trav.tyTrav.tyBtnGoToMag3.bValue					:= FALSE;
		tyP0936Trav.tyTrav.tyBtnGoToMag3.bRtLk					:= FALSE;
		tyP0936Trav.tyTrav.tyBtnGoToMag3.uiMaskRtStat.0			:= FALSE;

		tyP0936Trav.tyTrav.tyBtnGoToMag4.bRtCompl				:= FALSE;
		tyP0936Trav.tyTrav.tyBtnGoToMag4.bValue					:= FALSE;
		tyP0936Trav.tyTrav.tyBtnGoToMag4.bRtLk					:= FALSE;
		tyP0936Trav.tyTrav.tyBtnGoToMag4.uiMaskRtStat.0			:= FALSE;

		tyP0936Trav.tyMotionStd.tyBtnPwr.bRtCompl				:= FALSE;
		tyP0936Trav.tyMotionStd.tyBtnStop.bRtCompl				:= FALSE;
		tyP0936Trav.tyMotionStd.tyBtnOrigin.bRtCompl			:= FALSE;
		tyP0936Trav.tyMotionStd.tyBtnRst.bRtCompl				:= FALSE;
		tyP0936Trav.tyMotionStd.tyBtnMovAbs.bRtCompl			:= FALSE;
		tyP0936Trav.tyMotionStd.tyBtnMovRel.bRtCompl			:= FALSE;
		tyP0936Trav.tyMotionStd.tyBtnJogFront.bRtCompl			:= FALSE;
		tyP0936Trav.tyMotionStd.tyBtnJogRear.bRtCompl			:= FALSE;

		tyP0936Trav.tyMotionStd.tyBtnPwr.bValue					:= FALSE;
		tyP0936Trav.tyMotionStd.tyBtnStop.bValue				:= TRUE;
		tyP0936Trav.tyMotionStd.tyBtnOrigin.bValue				:= FALSE;
		tyP0936Trav.tyMotionStd.tyBtnRst.bValue					:= FALSE;
		tyP0936Trav.tyMotionStd.tyBtnMovAbs.bValue				:= FALSE;
		tyP0936Trav.tyMotionStd.tyBtnMovRel.bValue				:= FALSE;
		tyP0936Trav.tyMotionStd.tyBtnJogFront.bValue			:= FALSE;
		tyP0936Trav.tyMotionStd.tyBtnJogRear.bValue				:= FALSE;

		tyP0936Trav.tyMotionStd.tyBtnPwr.bRtLk					:= FALSE;
		tyP0936Trav.tyMotionStd.tyBtnStop.bRtLk					:= TRUE;
		tyP0936Trav.tyMotionStd.tyBtnOrigin.bRtLk				:= FALSE;
		tyP0936Trav.tyMotionStd.tyBtnRst.bRtLk					:= FALSE;
		tyP0936Trav.tyMotionStd.tyBtnMovAbs.bRtLk				:= FALSE;
		tyP0936Trav.tyMotionStd.tyBtnMovRel.bRtLk				:= FALSE;
		tyP0936Trav.tyMotionStd.tyBtnJogFront.bRtLk				:= FALSE;
		tyP0936Trav.tyMotionStd.tyBtnJogRear.bRtLk				:= FALSE;

		tyP0936Trav.tyMotionStd.tyBtnPwr.uiMaskRtStat			:= TRUE;
		tyP0936Trav.tyMotionStd.tyBtnOrigin.uiMaskRtStat		:= FALSE;
		tyP0936Trav.tyMotionStd.tyBtnRst.uiMaskRtStat			:= TRUE;
		tyP0936Trav.tyMotionStd.tyBtnMovAbs.uiMaskRtStat		:= FALSE;
		tyP0936Trav.tyMotionStd.tyBtnMovRel.uiMaskRtStat		:= FALSE;
		tyP0936Trav.tyMotionStd.tyBtnJogFront.uiMaskRtStat		:= FALSE;
		tyP0936Trav.tyMotionStd.tyBtnJogRear.uiMaskRtStat		:= FALSE;

	END_IF

	eInShutterAct	:= PneuActIdle;
	eOutShutterAct	:= PneuActIdle;

	tyP0936Trav.tyInOutletShutterFB.tyBtnClose.bRtCompl	:= FALSE;
	tyP0936Trav.tyInOutletShutterFB.tyBtnClose.bValue	:= FALSE;
	tyP0936Trav.tyInOutletShutterFB.tyBtnOpen.bRtCompl	:= FALSE;
	tyP0936Trav.tyInOutletShutterFB.tyBtnOpen.bValue	:= FALSE;

END_ACTION
```

#### Act_OptP0936UpdtDat.st
```iecst
ACTION Act_OptP0936UpdtDat:

	tyP0936Trav.tyMotionStd.tyNumCurrPos.diValue		:= p_diTravActualPos;
	tyP0936Trav.tyMotionStd.tyNumErrCode.diValue		:= UDINT_TO_DINT(p_udiTravAxisErrID);
	tyP0936Trav.tyMotionStd.tyBitmapPwr.usiValueIdx		:= BOOL_TO_USINT(p_bTravPwrOn);
	tyP0936Trav.tyMotionStd.tyBitmapRst.usiValueIdx		:= BOOL_TO_USINT(NOT p_bTravAxisErr);
	tyP0936Trav.tyMotionStd.tyBitmapOrigin.usiValueIdx	:= BOOL_TO_USINT(p_bTravIsHomed);
	tyP0936Trav.tyMotionStd.tyBtnFrontLmtSen.bValue		:= p_bTravFrontSen;
	tyP0936Trav.tyMotionStd.tyBtnRearLmtSen.bValue		:= p_bTravRearSen;

	//Machine Bitmap
	IF   (p_tyNtParamCurr.eProjMag = LDMagDual AND p_tyNtParamCurr.bMagAutoVerifyPrep = FALSE)
		OR (p_tyNtParamCurr.eProjMag = LDMagTriple AND p_tyNtParamCurr.bMagAutoVerifyPrep = FALSE)
		OR (p_tyNtParamCurr.eProjMag = LDMagDual AND p_tyNtParamCurr.bMagAutoVerifyPrep = TRUE)
		THEN
			IF p_bTravIsHomed = TRUE THEN
				IF p_diTravActualPos <= (p_tyNtParamCurr.tyUITravTargetPos.diMax / 3) THEN
					tyP0936Trav.tyMotionStd.tyBitmapMc.uiValueIdx 	:= 5;
				ELSIF p_diTravActualPos <= (p_tyNtParamCurr.tyUITravTargetPos.diMax / 3 * 2) THEN
					tyP0936Trav.tyMotionStd.tyBitmapMc.uiValueIdx 	:= 6;
				ELSE
					tyP0936Trav.tyMotionStd.tyBitmapMc.uiValueIdx 	:= 7;
				END_IF
			ELSE
				tyP0936Trav.tyMotionStd.tyBitmapMc.uiValueIdx	:= 5;
		END_IF

	ELSIF p_tyNtParamCurr.eProjMag = LDMagTriple AND p_tyNtParamCurr.bMagAutoVerifyPrep = TRUE
		THEN
			IF p_bTravIsHomed = TRUE THEN
				IF p_diTravActualPos <= (p_tyNtParamCurr.tyUITravTargetPos.diMax / 3) THEN
					tyP0936Trav.tyMotionStd.tyBitmapMc.uiValueIdx 	:= 26;
				ELSIF p_diTravActualPos <= (p_tyNtParamCurr.tyUITravTargetPos.diMax / 3 * 2) THEN
					tyP0936Trav.tyMotionStd.tyBitmapMc.uiValueIdx 	:= 27;
				ELSE
					tyP0936Trav.tyMotionStd.tyBitmapMc.uiValueIdx 	:= 28;
				END_IF
			ELSE
				tyP0936Trav.tyMotionStd.tyBitmapMc.uiValueIdx	:= 26;
			END_IF
	ELSIF p_tyNtParamCurr.eProjMag = LDMagQuadruple
		THEN
		IF p_bTravIsHomed = TRUE THEN
			IF p_diTravActualPos <= (p_tyNtParamCurr.tyUITravTargetPos.diMax / 3) THEN
				tyP0936Trav.tyMotionStd.tyBitmapMc.uiValueIdx 	:= 45;
			ELSIF p_diTravActualPos <= (p_tyNtParamCurr.tyUITravTargetPos.diMax / 3 * 2) THEN
				tyP0936Trav.tyMotionStd.tyBitmapMc.uiValueIdx 	:= 46;
			ELSE
				tyP0936Trav.tyMotionStd.tyBitmapMc.uiValueIdx 	:= 47;
			END_IF
		ELSE
			tyP0936Trav.tyMotionStd.tyBitmapMc.uiValueIdx	:= 45;
		END_IF
	END_IF

	IF p_tyNtParamCurr.eProjMag = LDMagTriple AND p_tyNtParamCurr.bProjLifterMagPlatform THEN
		IF 	tyP0936Trav.tyMotionStd.tyBitmapMc.uiValueIdx < 400 THEN
			tyP0936Trav.tyMotionStd.tyBitmapMc.uiValueIdx	:= tyP0936Trav.tyMotionStd.tyBitmapMc.uiValueIdx + 400;
		END_IF
	ELSIF p_tyNtParamCurr.eProjMag = LDMagTriple AND p_tyNtParamCurr.bMagAutoVerifyPrep = FALSE AND p_tyNtParamCurr.bProjMotorizedPullerPrep = FALSE AND p_tyNtParamCurr.bProjTopToBtmDefault = TRUE THEN
		IF 	tyP0936Trav.tyMotionStd.tyBitmapMc.uiValueIdx < 100 THEN
			tyP0936Trav.tyMotionStd.tyBitmapMc.uiValueIdx	:= tyP0936Trav.tyMotionStd.tyBitmapMc.uiValueIdx + 100;
		END_IF
	ELSIF p_tyNtParamCurr.eProjMag = LDMagTriple AND p_tyNtParamCurr.bMagAutoVerifyPrep = FALSE AND p_tyNtParamCurr.bProjMotorizedPullerPrep = FALSE AND p_tyNtParamCurr.bProjTopToBtmDefault = FALSE THEN
		IF 	tyP0936Trav.tyMotionStd.tyBitmapMc.uiValueIdx < 100 THEN
			tyP0936Trav.tyMotionStd.tyBitmapMc.uiValueIdx	:= tyP0936Trav.tyMotionStd.tyBitmapMc.uiValueIdx + 305-5;
		END_IF
	ELSIF p_tyNtParamCurr.eProjMag = LDMagDual AND p_tyNtParamCurr.bMagAutoVerifyPrep = FALSE THEN
		IF 	tyP0936Trav.tyMotionStd.tyBitmapMc.uiValueIdx < 100 THEN
			IF p_tyNtParamCurr.bProjLifterMagPlatform THEN
				//5,6,7
			ELSE
				IF p_tyNtParamCurr.sJobNo = '2023-0258A01' THEN
					tyP0936Trav.tyMotionStd.tyBitmapMc.uiValueIdx	:= tyP0936Trav.tyMotionStd.tyBitmapMc.uiValueIdx + 447-5;
				ELSIF p_tyNtParamCurr.sJobNo = '2023-0276A01' THEN
					tyP0936Trav.tyMotionStd.tyBitmapMc.uiValueIdx	:= tyP0936Trav.tyMotionStd.tyBitmapMc.uiValueIdx + 477-5;
				ELSE
					tyP0936Trav.tyMotionStd.tyBitmapMc.uiValueIdx	:= tyP0936Trav.tyMotionStd.tyBitmapMc.uiValueIdx + 200; //travLif
				END_IF

			END_IF
		END_IF
	ELSIF (p_tyNtParamCurr.eProjMag = LDMagDual OR p_tyNtParamCurr.eProjMag = LDMagTriple)
		AND p_tyNtParamCurr.bMagAutoVerifyPrep = TRUE THEN
			IF 	tyP0936Trav.tyMotionStd.tyBitmapMc.uiValueIdx < 200 THEN
				tyP0936Trav.tyMotionStd.tyBitmapMc.uiValueIdx	:= tyP0936Trav.tyMotionStd.tyBitmapMc.uiValueIdx + 200;
		END_IF
	ELSIF p_tyNtParamCurr.eProjMag = LDMagTriple AND p_tyNtParamCurr.bMagAutoVerifyPrep = FALSE AND p_tyNtParamCurr.bProjMotorizedPullerPrep = TRUE
		AND p_tyNtParamCurr.bProjCurtainSenPrep = FALSE THEN
		IF 	tyP0936Trav.tyMotionStd.tyBitmapMc.uiValueIdx < 300 THEN
			tyP0936Trav.tyMotionStd.tyBitmapMc.uiValueIdx	:= tyP0936Trav.tyMotionStd.tyBitmapMc.uiValueIdx + 300;
		END_IF
	ELSIF p_tyNtParamCurr.eProjMag = LDMagTriple AND p_tyNtParamCurr.bMagAutoVerifyPrep = FALSE AND p_tyNtParamCurr.bProjMotorizedPullerPrep = TRUE
		AND p_tyNtParamCurr.bProjCurtainSenPrep = TRUE AND p_tyNtParamCurr.bProjTopToBtmDefault = TRUE THEN
		IF 	tyP0936Trav.tyMotionStd.tyBitmapMc.uiValueIdx < 370-5 THEN
			tyP0936Trav.tyMotionStd.tyBitmapMc.uiValueIdx	:= tyP0936Trav.tyMotionStd.tyBitmapMc.uiValueIdx + 370-5;
		END_IF
	ELSIF p_tyNtParamCurr.eProjMag = LDMagTriple AND p_tyNtParamCurr.bMagAutoVerifyPrep = FALSE AND p_tyNtParamCurr.bProjMotorizedPullerPrep = TRUE
		AND p_tyNtParamCurr.bProjCurtainSenPrep = TRUE AND p_tyNtParamCurr.bProjTopToBtmDefault = FALSE THEN
		IF 	tyP0936Trav.tyMotionStd.tyBitmapMc.uiValueIdx < 423-5 THEN
			tyP0936Trav.tyMotionStd.tyBitmapMc.uiValueIdx	:= tyP0936Trav.tyMotionStd.tyBitmapMc.uiValueIdx + 423-5;
		END_IF
	END_IF
END_ACTION
```

#### Act_EntP0937Disp.st
```iecst
ACTION Act_EntP0937Disp:

	// Access Address
	p_tyC0001MotionStd ACCESS ADR(tyP0937AWPushOrPuller.tyMotionStd);

	p_tyC0002FullMask ACCESS ADR(tyP0937AWPushOrPuller.tyFullMaskHide);

	p_tyC0004Navi ACCESS ADR(tyP0937AWPushOrPuller.tyNaviBack);

	p_tyC0005Main ACCESS ADR(tyCommon.tyMain);

	p_tyC0007Notif ACCESS ADR(tyCommon.tyNotif);

	p_tyC0008MsgBox ACCESS ADR(tyP0937AWPushOrPuller.tyMsgBoxHide);

	p_tyC0009Info ACCESS ADR(tyCommon.tyInfo);

	p_tyP0937AWPushOrPuller ACCESS ADR(tyP0937AWPushOrPuller.tyAW);
	p_tyP0937InOutletShutterFB ACCESS ADR(tyP0937AWPushOrPuller.tyInOutletShutterFB);

	// Display
	tyP0937AWPushOrPuller.tyAW.tyNumNewWidth.diValue		:= p_tyProdRcpCurrRcp0.diWidthInUM;

	tyP0937AWPushOrPuller.tyMotionStd.tyBtnPwr.bValue		:= p_bAWPushOrPullerPwrOn;

	fbLmtRstTm(IN := FALSE);

END_ACTION
```
